      BB_G2_KS_AM19 : Bool;   // Belebung - SigmaControl Gebläse 2 - Alarme - Ansaugdruck p1 zu niedrig -> Verschmutzung des Ansaugfilters
      BB_G2_KS_AM20 : Bool;   // Belebung - SigmaControl Gebläse 2 - Alarme - Temperatur unter der Schalldämmhaube zu hoch
      BB_G2_KS_AM21 : Bool;   // Belebung - SigmaControl Gebläse 2 - Alarme - Reserve
      BB_G2_KS_AM22 : Bool;   // Belebung - SigmaControl Gebläse 2 - Alarme - Differenzdruck zu hoch
      BB_G2_KS_AM23 : Bool;   // Belebung - SigmaControl Gebläse 2 - Alarme - Ansaugtemperatur t1 zu hoch
      BB_G2_KS_AM24 : Bool;   // Belebung - SigmaControl Gebläse 2 - Alarme - Ansaugtemperatur t1 zu niedrig
      BB_G2_KS_AM41 : Bool;   // Belebung - SigmaControl Gebläse 2 - Alarme - Überspannung im Stromversorgungsnetz
      BB_G2_KS_AM42 : Bool;   // Belebung - SigmaControl Gebläse 2 - Alarme - Fehler am AFxM-Ventil-Aktor
      BB_G2_KS_AM43 : Bool;   // Belebung - SigmaControl Gebläse 2 - Alarme - Reserve
      BB_G2_KS_AM44 : Bool;   // Belebung - SigmaControl Gebläse 2 - Alarme - Blockdrehzahl liegt außerhalb des erlaubten Bereiches -> Fehler im Antriebsmotor oder Keilriemen
      BB_G2_KS_AM45 : Bool;   // Belebung - SigmaControl Gebläse 2 - Alarme - Vibration des Gebläses zu hoch
      BB_G2_KS_AM46 : Bool;   // Belebung - SigmaControl Gebläse 2 - Alarme - Interner Fehler Frequenzumrichter für Gebläsemotor
      BB_G2_KS_AM47 : Bool;   // Belebung - SigmaControl Gebläse 2 - Alarme - Kommunikationsfehler RS485-FC -> USS-Bus Kommunikationsfehler
      BB_G2_KS_AM48 : Bool;   // Belebung - SigmaControl Gebläse 2 - Alarme - Sammelmeldung des Leistungsteils FU
      BB_G2_KS_AM33 : Bool;   // Belebung - SigmaControl Gebläse 2 - Alarme - Reserve
      BB_G2_KS_AM34 : Bool;   // Belebung - SigmaControl Gebläse 2 - Alarme - Reserve
      BB_G2_KS_AM35 : Bool;   // Belebung - SigmaControl Gebläse 2 - Alarme - Druckdifferenz über den Block zu niedrig
      BB_G2_KS_AM36 : Bool;   // Belebung - SigmaControl Gebläse 2 - Alarme - Reserve
      BB_G2_KS_AM37 : Bool;   // Belebung - SigmaControl Gebläse 2 - Alarme - Reserve
      BB_G2_KS_AM38 : Bool;   // Belebung - SigmaControl Gebläse 2 - Alarme - Ansaugdruck p1 zu niedrig -> Verschmutzung des Ansaugfilters
      BB_G2_KS_AM39 : Bool;   // Belebung - SigmaControl Gebläse 2 - Alarme - Enddruck p2 zu hoch
      BB_G2_KS_AM40 : Bool;   // Belebung - SigmaControl Gebläse 2 - Alarme - Netzschütz schaltet nicht aus oder nicht ein
      BB_G2_KS_AM57 : Bool;   // Belebung - SigmaControl Gebläse 2 - Alarme - Schwerlastüberwachung ausgelöst FU -> Schwerlastüberwachung ausgelöst
      BB_G2_KS_AM58 : Bool;   // Belebung - SigmaControl Gebläse 2 - Alarme - p1-Sensor-Fehler Fehler Drucksensor Ansaugseite Gebläseblock
      BB_G2_KS_AM59 : Bool;   // Belebung - SigmaControl Gebläse 2 - Alarme - p2-Sensor-Fehler Fehler Drucksensor Auslassseite Gebläseblock
      BB_G2_KS_AM60 : Bool;   // Belebung - SigmaControl Gebläse 2 - Alarme - Fehler externer Analogeingang Fehler am externen Analogeingang
      BB_G2_KS_AM61 : Bool;   // Belebung - SigmaControl Gebläse 2 - Alarme - t2-Sensor-Fehler Fehler Sensor PT100 Auslasssseite Gebläseblock
      BB_G2_KS_AM62 : Bool;   // Belebung - SigmaControl Gebläse 2 - Alarme - t_S-Sensor-Fehler Fehler Sensor PT100 Schalldämmhaube
      BB_G2_KS_AM63 : Bool;   // Belebung - SigmaControl Gebläse 2 - Alarme - t1-Sensor-Fehler Fehler Sensor PT100 Ansaugseite Gebläseblock
      BB_G2_KS_AM64 : Bool;   // Belebung - SigmaControl Gebläse 2 - Alarme - t_M-Sensor-Fehler Fehler Sensor PT100 Antriebsmotor
      BB_G2_KS_AM49 : Bool;   // Belebung - SigmaControl Gebläse 2 - Alarme - Reserve
      BB_G2_KS_AM50 : Bool;   // Belebung - SigmaControl Gebläse 2 - Alarme - Nachschmiereinrichtung meldet seit längerer Zeit einen Fehler
      BB_G2_KS_AM51 : Bool;   // Belebung - SigmaControl Gebläse 2 - Alarme - Reserve
      BB_G2_KS_AM52 : Bool;   // Belebung - SigmaControl Gebläse 2 - Alarme - Reserve
      BB_G2_KS_AM53 : Bool;   // Belebung - SigmaControl Gebläse 2 - Alarme - Fehler USS Handler FU -> USS Busfehler
      BB_G2_KS_AM54 : Bool;   // Belebung - SigmaControl Gebläse 2 - Alarme - PKW-Anfragen erfolglos FU -> USS Kommunikation gestört
      BB_G2_KS_AM55 : Bool;   // Belebung - SigmaControl Gebläse 2 - Alarme - Fehler FU Einschaltung FU -> Fehler beim Einschalten des Frequenzumrichters
      BB_G2_KS_AM56 : Bool;   // Belebung - SigmaControl Gebläse 2 - Alarme - Motor -> n_min nicht erreicht FU -> Mindestdrehzahl nicht erreicht
      BB_G2_KS_AM73 : Bool;   // Belebung - SigmaControl Gebläse 2 - Alarme - Externe Meldung 1 Sammelmeldung externe Binärmeldung 1
      BB_G2_KS_AM74 : Bool;   // Belebung - SigmaControl Gebläse 2 - Alarme - Externe Meldung 2 Sammelmeldung externe Binärmeldung 2
      BB_G2_KS_AM75 : Bool;   // Belebung - SigmaControl Gebläse 2 - Alarme - Externe Meldung 3 Sammelmeldung externe Binärmeldung 3
      BB_G2_KS_AM76 : Bool;   // Belebung - SigmaControl Gebläse 2 - Alarme - Schalter p1 freier Schaltpunkt auf Druck p1
      BB_G2_KS_AM77 : Bool;   // Belebung - SigmaControl Gebläse 2 - Alarme - Schalter p2 freier Schaltpunkt auf Druck p2
      BB_G2_KS_AM78 : Bool;   // Belebung - SigmaControl Gebläse 2 - Alarme - Schalter T1 freier Schaltpunkt auf Temperatur T1
      BB_G2_KS_AM79 : Bool;   // Belebung - SigmaControl Gebläse 2 - Alarme - Schalter T2 freier Schaltpunkt auf Temperatur T2
      BB_G2_KS_AM80 : Bool;   // Belebung - SigmaControl Gebläse 2 - Alarme - Schalter Blockdrehzahl freier Schaltpunkt auf Blockdrehzahl
      BB_G2_KS_AM65 : Bool;   // Belebung - SigmaControl Gebläse 2 - Alarme - t3-Sensor-Fehler Fehler Sensor PT100 Öltemperatur
      BB_G2_KS_AM66 : Bool;   // Belebung - SigmaControl Gebläse 2 - Alarme - Reserve
      BB_G2_KS_AM67 : Bool;   // Belebung - SigmaControl Gebläse 2 - Alarme - Reserve
      BB_G2_KS_AM68 : Bool;   // Belebung - SigmaControl Gebläse 2 - Alarme - Reserve
      BB_G2_KS_AM69 : Bool;   // Belebung - SigmaControl Gebläse 2 - Alarme - Reserve
      BB_G2_KS_AM70 : Bool;   // Belebung - SigmaControl Gebläse 2 - Alarme - Schwingungsüberwachung VSE ? Schwingungen an Block oder Motor zu hoch
      BB_G2_KS_AM71 : Bool;   // Belebung - SigmaControl Gebläse 2 - Alarme - Schalter T3
      BB_G2_KS_AM72 : Bool;   // Belebung - SigmaControl Gebläse 2 - Alarme - Schalter T_S
      BB_G2_KS_WM9 : Bool;   // Belebung - SigmaControl Gebläse 2 - Warnungen - Temperatur unter der Schalldämmhaube zu hoch
      BB_G2_KS_WM10 : Bool;   // Belebung - SigmaControl Gebläse 2 - Warnungen - Umgebungstemperatur zu niedrig
      BB_G2_KS_WM11 : Bool;   // Belebung - SigmaControl Gebläse 2 - Warnungen - Differenzdruck zu hoch
      BB_G2_KS_WM12 : Bool;   // Belebung - SigmaControl Gebläse 2 - Warnungen - Differenzdruck zu niedrig
      BB_G2_KS_WM13 : Bool;   // Belebung - SigmaControl Gebläse 2 - Warnungen - Filter verstopft, Verschmutzung des Ansaugfilters
      BB_G2_KS_WM14 : Bool;   // Belebung - SigmaControl Gebläse 2 - Warnungen - Öltemperatur t3 zu hoch
      BB_G2_KS_WM15 : Bool;   // Belebung - SigmaControl Gebläse 2 - Warnungen - Com-Module Kommunikationsfehler Busankopplung über Com-Module ist unterbrochen
      BB_G2_KS_WM16 : Bool;   // Belebung - SigmaControl Gebläse 2 - Warnungen - SAM 4.0 Kommunikationsfehler Busankopplung über Com-Module ist unterbrochen
      BB_G2_KS_WM1 : Bool;   // Belebung - SigmaControl Gebläse 2 - Warnungen - Equipmentnummer unvollständig -> Equipmentnummer des Gebläses hat weniger als sieben Zeichen
      BB_G2_KS_WM2 : Bool;   // Belebung - SigmaControl Gebläse 2 - Warnungen - Sammelwarnung
      BB_G2_KS_WM3 : Bool;   // Belebung - SigmaControl Gebläse 2 - Warnungen - Reserve
      BB_G2_KS_WM4 : Bool;   // Belebung - SigmaControl Gebläse 2 - Warnungen - Schmierölstand Antriebsseite Gebläseblock zu niedrig
      BB_G2_KS_WM5 : Bool;   // Belebung - SigmaControl Gebläse 2 - Warnungen - Schmierölstand Steuerseite Gebläseblock zu niedrig
      BB_G2_KS_WM6 : Bool;   // Belebung - SigmaControl Gebläse 2 - Warnungen - Ansaugtemperatur t1 zu hoch
      BB_G2_KS_WM7 : Bool;   // Belebung - SigmaControl Gebläse 2 - Warnungen - Ansaugtemperatur t1 zu niedrig
      BB_G2_KS_WM8 : Bool;   // Belebung - SigmaControl Gebläse 2 - Warnungen - Verdichtungsendtemperatur t2 zu hoch
      BB_G2_KS_WM25 : Bool;   // Belebung - SigmaControl Gebläse 2 - Warnungen - Motorlager Schaltschrank-Lüfter -> Prüffrist abgelaufen
      BB_G2_KS_WM26 : Bool;   // Belebung - SigmaControl Gebläse 2 - Warnungen - Schmieröl -> Wartungsfrist abgelaufen
      BB_G2_KS_WM27 : Bool;   // Belebung - SigmaControl Gebläse 2 - Warnungen - Reserve
      BB_G2_KS_WM28 : Bool;   // Belebung - SigmaControl Gebläse 2 - Warnungen - Ansaugluftfilter -> Wartungsfrist abgelaufen
      BB_G2_KS_WM29 : Bool;   // Belebung - SigmaControl Gebläse 2 - Warnungen - Filtermatte -> Wartungsfrist abgelaufen
      BB_G2_KS_WM30 : Bool;   // Belebung - SigmaControl Gebläse 2 - Warnungen - Keilriemen -> Wartungsfrist abgelaufen
      BB_G2_KS_WM31 : Bool;   // Belebung - SigmaControl Gebläse 2 - Warnungen - Motorlager -> Wartungsfrist abgelaufen
      BB_G2_KS_WM32 : Bool;   // Belebung - SigmaControl Gebläse 2 - Warnungen - Motorlager Gebläsemotor -> Prüffrist abgelaufen
      BB_G2_KS_WM17 : Bool;   // Belebung - SigmaControl Gebläse 2 - Warnungen - Temperaturdifferenz t2 (VET) - t1 (Ansaugtemperatur) zu hoch
      BB_G2_KS_WM18 : Bool;   // Belebung - SigmaControl Gebläse 2 - Warnungen - Temperatur Gebläsemotor zu hoch
      BB_G2_KS_WM19 : Bool;   // Belebung - SigmaControl Gebläse 2 - Warnungen - Ansaugdruck p1 zu niedrig -> Verschmutzung des Ansaugfilters
      BB_G2_KS_WM20 : Bool;   // Belebung - SigmaControl Gebläse 2 - Warnungen - Enddruck p2 zu hoch
      BB_G2_KS_WM21 : Bool;   // Belebung - SigmaControl Gebläse 2 - Warnungen - Öltemperatur t3 zu niedrig
      BB_G2_KS_WM22 : Bool;   // Belebung - SigmaControl Gebläse 2 - Warnungen - Druckverhältnis über Block zu hoch
      BB_G2_KS_WM23 : Bool;   // Belebung - SigmaControl Gebläse 2 - Warnungen - Reserve
      BB_G2_KS_WM24 : Bool;   // Belebung - SigmaControl Gebläse 2 - Warnungen - maximale Schalthäufigkeit des Netzschützes ist erreicht -> austauschen
      BB_G2_KS_WM41 : Bool;   // Belebung - SigmaControl Gebläse 2 - Warnungen - Reserve
      BB_G2_KS_WM42 : Bool;   // Belebung - SigmaControl Gebläse 2 - Warnungen - Reserve
      BB_G2_KS_WM43 : Bool;   // Belebung - SigmaControl Gebläse 2 - Warnungen - Reserve
      BB_G2_KS_WM44 : Bool;   // Belebung - SigmaControl Gebläse 2 - Warnungen - Reserve
      BB_G2_KS_WM45 : Bool;   // Belebung - SigmaControl Gebläse 2 - Warnungen - Reserve
      BB_G2_KS_WM46 : Bool;   // Belebung - SigmaControl Gebläse 2 - Warnungen - Reserve
      BB_G2_KS_WM47 : Bool;   // Belebung - SigmaControl Gebläse 2 - Warnungen - Elektrobauteile und -installation -> Wartungsfrist abgelaufen
      BB_G2_KS_WM48 : Bool;   // Belebung - SigmaControl Gebläse 2 - Warnungen - Schmierung Motorlager Gebläsemotor -> Wartungsfrist abgelaufen
      BB_G2_KS_WM33 : Bool;   // Belebung - SigmaControl Gebläse 2 - Warnungen - Motorlager Schalldämmhauben-Lüfter -> Prüffrist abgelaufen
      BB_G2_KS_WM34 : Bool;   // Belebung - SigmaControl Gebläse 2 - Warnungen - FU-Lüfter -> Prüffrist abgelaufen
      BB_G2_KS_WM35 : Bool;   // Belebung - SigmaControl Gebläse 2 - Warnungen - Filter Getriebeentlüftung -> Wartungsfrist abgelaufen
      BB_G2_KS_WM36 : Bool;   // Belebung - SigmaControl Gebläse 2 - Warnungen - Maximal zulässige Schalthäufigkeit des Motors in den letzten 60 Minuten überschritten
      BB_G2_KS_WM37 : Bool;   // Belebung - SigmaControl Gebläse 2 - Warnungen - Reserve
      BB_G2_KS_WM38 : Bool;   // Belebung - SigmaControl Gebläse 2 - Warnungen - Ansaugdruck p1 zu niedrig -> Verschmutzung des Ansaugfilters
      BB_G2_KS_WM39 : Bool;   // Belebung - SigmaControl Gebläse 2 - Warnungen - Enddruck p2 zu hoch
      BB_G2_KS_WM40 : Bool;   // Belebung - SigmaControl Gebläse 2 - Warnungen - Überspannung im Stromversorgungsnetz
      BB_G2_KS_WM57 : Bool;   // Belebung - SigmaControl Gebläse 2 - Warnungen - Reserve
      BB_G2_KS_WM58 : Bool;   // Belebung - SigmaControl Gebläse 2 - Warnungen - SC2 zu SC2 Kommunikation unterbrochen
      BB_G2_KS_WM59 : Bool;   // Belebung - SigmaControl Gebläse 2 - Warnungen - Reserve
      BB_G2_KS_WM60 : Bool;   // Belebung - SigmaControl Gebläse 2 - Warnungen - Reserve
      BB_G2_KS_WM61 : Bool;   // Belebung - SigmaControl Gebläse 2 - Warnungen - Reserve
      BB_G2_KS_WM62 : Bool;   // Belebung - SigmaControl Gebläse 2 - Warnungen - FU im Servicebetrieb
      BB_G2_KS_WM63 : Bool;   // Belebung - SigmaControl Gebläse 2 - Warnungen - Test der "Safe Torque off" Abschaltpfade des Frequenzumrichters
      BB_G2_KS_WM64 : Bool;   // Belebung - SigmaControl Gebläse 2 - Warnungen - Reserve
      BB_G2_KS_WM49 : Bool;   // Belebung - SigmaControl Gebläse 2 - Warnungen - Jahreswartung fällig (erscheint 1 Jahr nach letzter Wartung)
      BB_G2_KS_WM50 : Bool;   // Belebung - SigmaControl Gebläse 2 - Warnungen - Fehler beim Schreiben der Daten auf SD-Karte
      BB_G2_KS_WM51 : Bool;   // Belebung - SigmaControl Gebläse 2 - Warnungen - Nachschmiereinrichtung meldet einen Fehler
      BB_G2_KS_WM52 : Bool;   // Belebung - SigmaControl Gebläse 2 - Warnungen - Reserve
      BB_G2_KS_WM53 : Bool;   // Belebung - SigmaControl Gebläse 2 - Warnungen - Reserve
      BB_G2_KS_WM54 : Bool;   // Belebung - SigmaControl Gebläse 2 - Warnungen - Reserve
      BB_G2_KS_WM55 : Bool;   // Belebung - SigmaControl Gebläse 2 - Warnungen - Reserve
      BB_G2_KS_WM56 : Bool;   // Belebung - SigmaControl Gebläse 2 - Warnungen - Reserve
      BB_G2_KS_WM73 : Bool;   // Belebung - SigmaControl Gebläse 2 - Warnungen - Sammelmeldung externe Binärmeldung 1
      BB_G2_KS_WM74 : Bool;   // Belebung - SigmaControl Gebläse 2 - Warnungen - Sammelmeldung externe Binärmeldung 2
      BB_G2_KS_WM75 : Bool;   // Belebung - SigmaControl Gebläse 2 - Warnungen - Sammelmeldung externe Binärmeldung 3
      BB_G2_KS_WM76 : Bool;   // Belebung - SigmaControl Gebläse 2 - Warnungen - Schalter p1 freier Schaltpunkt auf Druck p1
      BB_G2_KS_WM77 : Bool;   // Belebung - SigmaControl Gebläse 2 - Warnungen - Schalter p2 freier Schaltpunkt auf Druck p2
      BB_G2_KS_WM78 : Bool;   // Belebung - SigmaControl Gebläse 2 - Warnungen - Schalter T1 freier Schaltpunkt auf Temperatur T1
      BB_G2_KS_WM79 : Bool;   // Belebung - SigmaControl Gebläse 2 - Warnungen - Schalter T2 freier Schaltpunkt auf Temperatur T2
      BB_G2_KS_WM80 : Bool;   // Belebung - SigmaControl Gebläse 2 - Warnungen - Schalter Blockdrehzahl freier Schaltpunkt auf Blockdrehzahl
      BB_G2_KS_WM65 : Bool;   // Belebung - SigmaControl Gebläse 2 - Warnungen - Reserve
      BB_G2_KS_WM66 : Bool;   // Belebung - SigmaControl Gebläse 2 - Warnungen - Reserve
      BB_G2_KS_WM67 : Bool;   // Belebung - SigmaControl Gebläse 2 - Warnungen - Reserve
      BB_G2_KS_WM68 : Bool;   // Belebung - SigmaControl Gebläse 2 - Warnungen - Schalter T3
      BB_G2_KS_WM69 : Bool;   // Belebung - SigmaControl Gebläse 2 - Warnungen - Schalter T_S
      BB_G2_KS_WM70 : Bool;   // Belebung - SigmaControl Gebläse 2 - Warnungen - Schwingungsüberwachung VSE -> Schwingungen an Block oder Motor
      BB_G2_KS_WM71 : Bool;   // Belebung - SigmaControl Gebläse 2 - Warnungen - Schwingungsüberwachung VSE -> Schwingungen an Block oder Motor
      BB_G2_KS_WM72 : Bool;   // Belebung - SigmaControl Gebläse 2 - Warnungen - Schwingungsüberwachung Summensignal -> Schwingungen an Block oder Motor
      BB_G2_KS_OM9 : Bool;   // Belebung - SigmaControl Gebläse 2 - Betriebsmeldungen - Reserve
      BB_G2_KS_OM10 : Bool;   // Belebung - SigmaControl Gebläse 2 - Betriebsmeldungen - Reserve
      BB_G2_KS_OM11 : Bool;   // Belebung - SigmaControl Gebläse 2 - Betriebsmeldungen - Warten auf Kaltstart -> Temperaturen im Gebläse zu niedrig
      BB_G2_KS_OM12 : Bool;   // Belebung - SigmaControl Gebläse 2 - Betriebsmeldungen - Ölrücklauf vom Filter in die Ölräume gestartet
      BB_G2_KS_OM13 : Bool;   // Belebung - SigmaControl Gebläse 2 - Betriebsmeldungen - Ölmangel (Ölrücklauf abwarten, Ölstand zu niedrig)
      BB_G2_KS_OM14 : Bool;   // Belebung - SigmaControl Gebläse 2 - Betriebsmeldungen - Reserve
      BB_G2_KS_OM15 : Bool;   // Belebung - SigmaControl Gebläse 2 - Betriebsmeldungen - Reserve
      BB_G2_KS_OM16 : Bool;   // Belebung - SigmaControl Gebläse 2 - Betriebsmeldungen - Reserve
      BB_G2_KS_OM1 : Bool;   // Belebung - SigmaControl Gebläse 2 - Betriebsmeldungen - Reserve
      BB_G2_KS_OM2 : Bool;   // Belebung - SigmaControl Gebläse 2 - Betriebsmeldungen - Reserve
      BB_G2_KS_OM3 : Bool;   // Belebung - SigmaControl Gebläse 2 - Betriebsmeldungen - Reserve
      BB_G2_KS_OM4 : Bool;   // Belebung - SigmaControl Gebläse 2 - Betriebsmeldungen - Reserve
      BB_G2_KS_OM5 : Bool;   // Belebung - SigmaControl Gebläse 2 - Betriebsmeldungen - Reserve
      BB_G2_KS_OM6 : Bool;   // Belebung - SigmaControl Gebläse 2 - Betriebsmeldungen - Reserve
      BB_G2_KS_OM7 : Bool;   // Belebung - SigmaControl Gebläse 2 - Betriebsmeldungen - Reserve
      BB_G2_KS_OM8 : Bool;   // Belebung - SigmaControl Gebläse 2 - Betriebsmeldungen - Reserve
      BB_G2_KS_OM25 : Bool;   // Belebung - SigmaControl Gebläse 2 - Betriebsmeldungen - Reserve
      BB_G2_KS_OM26 : Bool;   // Belebung - SigmaControl Gebläse 2 - Betriebsmeldungen - Reserve
      BB_G2_KS_OM27 : Bool;   // Belebung - SigmaControl Gebläse 2 - Betriebsmeldungen - Power OFF -> ON Neustart der Steuerung erforderlich
      BB_G2_KS_OM28 : Bool;   // Belebung - SigmaControl Gebläse 2 - Betriebsmeldungen - Reserve
      BB_G2_KS_OM29 : Bool;   // Belebung - SigmaControl Gebläse 2 - Betriebsmeldungen - Reserve
      BB_G2_KS_OM30 : Bool;   // Belebung - SigmaControl Gebläse 2 - Betriebsmeldungen - Schalter p1 freier Schaltpunkt auf Druck p1
      BB_G2_KS_OM31 : Bool;   // Belebung - SigmaControl Gebläse 2 - Betriebsmeldungen - Schalter p2 freier Schaltpunkt auf Druck p2
      BB_G2_KS_OM32 : Bool;   // Belebung - SigmaControl Gebläse 2 - Betriebsmeldungen - Schalter T1 freier Schaltpunkt auf Temperatur T1
      BB_G2_KS_OM17 : Bool;   // Belebung - SigmaControl Gebläse 2 - Betriebsmeldungen - Externe Meldung 1 Sammelmeldung externe Binärmeldung 1
      BB_G2_KS_OM18 : Bool;   // Belebung - SigmaControl Gebläse 2 - Betriebsmeldungen - Externe Meldung 2 Sammelmeldung externe Binärmeldung 2
      BB_G2_KS_OM19 : Bool;   // Belebung - SigmaControl Gebläse 2 - Betriebsmeldungen - Externe Meldung 3 Sammelmeldung externe Binärmeldung 3
      BB_G2_KS_OM20 : Bool;   // Belebung - SigmaControl Gebläse 2 - Betriebsmeldungen - Schwingungsüberwachung VSE -> Schwingungen an Block oder Motor
      BB_G2_KS_OM21 : Bool;   // Belebung - SigmaControl Gebläse 2 - Betriebsmeldungen - Schwingungsüberwachung Summensignal -> Schwingungen an Block oder Motor
      BB_G2_KS_OM22 : Bool;   // Belebung - SigmaControl Gebläse 2 - Betriebsmeldungen - Reserve
      BB_G2_KS_OM23 : Bool;   // Belebung - SigmaControl Gebläse 2 - Betriebsmeldungen - Reserve
      BB_G2_KS_OM24 : Bool;   // Belebung - SigmaControl Gebläse 2 - Betriebsmeldungen - Reserve
      BB_G2_KS_OM41 : Bool;   // Belebung - SigmaControl Gebläse 2 - Betriebsmeldungen - Reserve
      BB_G2_KS_OM42 : Bool;   // Belebung - SigmaControl Gebläse 2 - Betriebsmeldungen - Reserve
      BB_G2_KS_OM43 : Bool;   // Belebung - SigmaControl Gebläse 2 - Betriebsmeldungen - Reserve
      BB_G2_KS_OM44 : Bool;   // Belebung - SigmaControl Gebläse 2 - Betriebsmeldungen - Reserve
      BB_G2_KS_OM45 : Bool;   // Belebung - SigmaControl Gebläse 2 - Betriebsmeldungen - Reserve
      BB_G2_KS_OM46 : Bool;   // Belebung - SigmaControl Gebläse 2 - Betriebsmeldungen - Reserve
      BB_G2_KS_OM47 : Bool;   // Belebung - SigmaControl Gebläse 2 - Betriebsmeldungen - Reserve
      BB_G2_KS_OM48 : Bool;   // Belebung - SigmaControl Gebläse 2 - Betriebsmeldungen - Reserve
      BB_G2_KS_OM33 : Bool;   // Belebung - SigmaControl Gebläse 2 - Betriebsmeldungen - Schalter T2 freier Schaltpunkt auf Temperatur T2
      BB_G2_KS_OM34 : Bool;   // Belebung - SigmaControl Gebläse 2 - Betriebsmeldungen - Schalter Blockdrehzahl freier Schaltpunkt auf Blockdrehzahl
      BB_G2_KS_OM35 : Bool;   // Belebung - SigmaControl Gebläse 2 - Betriebsmeldungen - Schalter T3
      BB_G2_KS_OM36 : Bool;   // Belebung - SigmaControl Gebläse 2 - Betriebsmeldungen - Schalter T_S
      BB_G2_KS_OM37 : Bool;   // Belebung - SigmaControl Gebläse 2 - Betriebsmeldungen - Reserve
      BB_G2_KS_OM38 : Bool;   // Belebung - SigmaControl Gebläse 2 - Betriebsmeldungen - Ansaugdruck p1 zu niedrig -> Verschmutzung des Ansaugfilters
      BB_G2_KS_OM39 : Bool;   // Belebung - SigmaControl Gebläse 2 - Betriebsmeldungen - Enddruck p2 zu hoch
      BB_G2_KS_OM40 : Bool;   // Belebung - SigmaControl Gebläse 2 - Betriebsmeldungen - Techniker vor Ort Ein Techniker arbeitet an der Maschine
      BB_G2_KS_BS8 : Bool;   // Belebung - SigmaControl Gebläse 2 - Status - Reserve
      BB_G2_KS_BS9 : Bool;   // Belebung - SigmaControl Gebläse 2 - Status - Gebläse Ein (Maschine eingeschaltet)
      BB_G2_KS_BS10 : Bool;   // Belebung - SigmaControl Gebläse 2 - Status - Lüfter Nachkühler Betrieb
      BB_G2_KS_BS11 : Bool;   // Belebung - SigmaControl Gebläse 2 - Status - Lüfter Schalldämmhaube Betrieb
      BB_G2_KS_BS12 : Bool;   // Belebung - SigmaControl Gebläse 2 - Status - Reserve
      BB_G2_KS_BS13 : Bool;   // Belebung - SigmaControl Gebläse 2 - Status - Reserve
      BB_G2_KS_BS14 : Bool;   // Belebung - SigmaControl Gebläse 2 - Status - Sammelwartung
      BB_G2_KS_BS15 : Bool;   // Belebung - SigmaControl Gebläse 2 - Status - Sammelwarnung
      BB_G2_KS_BS0 : Bool;   // Belebung - SigmaControl Gebläse 2 - Status - Anlage Ein + Fernbetrieb Ein + Bus (Receive)
      BB_G2_KS_BS1 : Bool;   // Belebung - SigmaControl Gebläse 2 - Status - Motor Betrieb
      BB_G2_KS_BS2 : Bool;   // Belebung - SigmaControl Gebläse 2 - Status - Lastlauf
      BB_G2_KS_BS3 : Bool;   // Belebung - SigmaControl Gebläse 2 - Status - Leerlauf
      BB_G2_KS_BS4 : Bool;   // Belebung - SigmaControl Gebläse 2 - Status - vor-Ort Betrieb
      BB_G2_KS_BS5 : Bool;   // Belebung - SigmaControl Gebläse 2 - Status - Anlage Ein
      BB_G2_KS_BS6 : Bool;   // Belebung - SigmaControl Gebläse 2 - Status - Sammelstörung
      BB_G2_KS_BS7 : Bool;   // Belebung - SigmaControl Gebläse 2 - Status - Sammelwarnung/-warnung
      BB_G2_KS_BS24 : Bool;   // Belebung - SigmaControl Gebläse 2 - Status - Betriebsart Volumenstromregelung
      BB_G2_KS_BS25 : Bool;   // Belebung - SigmaControl Gebläse 2 - Status - Reserve
      BB_G2_KS_BS26 : Bool;   // Belebung - SigmaControl Gebläse 2 - Status - Reserve
      BB_G2_KS_BS27 : Bool;   // Belebung - SigmaControl Gebläse 2 - Status - Reserve
      BB_G2_KS_BS28 : Bool;   // Belebung - SigmaControl Gebläse 2 - Status - Reserve
      BB_G2_KS_BS29 : Bool;   // Belebung - SigmaControl Gebläse 2 - Status - Reserve
      BB_G2_KS_BS30 : Bool;   // Belebung - SigmaControl Gebläse 2 - Status - Reserve
      BB_G2_KS_BS31 : Bool;   // Belebung - SigmaControl Gebläse 2 - Status - Reserve
      BB_G2_KS_BS16 : Bool;   // Belebung - SigmaControl Gebläse 2 - Status - Modus "Gebläse Ein" nur durch vor-Ort-Bedienung
      BB_G2_KS_BS17 : Bool;   // Belebung - SigmaControl Gebläse 2 - Status - Reserve
      BB_G2_KS_BS18 : Bool;   // Belebung - SigmaControl Gebläse 2 - Status - Reserve
      BB_G2_KS_BS19 : Bool;   // Belebung - SigmaControl Gebläse 2 - Status - Reserve
      BB_G2_KS_BS20 : Bool;   // Belebung - SigmaControl Gebläse 2 - Status - Betriebsart Festdrehzahl
      BB_G2_KS_BS21 : Bool;   // Belebung - SigmaControl Gebläse 2 - Status - Betriebsart externe Drehzahlvorgabe
      BB_G2_KS_BS22 : Bool;   // Belebung - SigmaControl Gebläse 2 - Status - Betriebsart Druckregelung
      BB_G2_KS_BS23 : Bool;   // Belebung - SigmaControl Gebläse 2 - Status - Betriebsart externe Größe
      BB_G2_KS_BS40 : Bool;   // Belebung - SigmaControl Gebläse 2 - Status - Reserve
      BB_G2_KS_BS41 : Bool;   // Belebung - SigmaControl Gebläse 2 - Status - Reserve
      BB_G2_KS_BS42 : Bool;   // Belebung - SigmaControl Gebläse 2 - Status - Reserve
      BB_G2_KS_BS43 : Bool;   // Belebung - SigmaControl Gebläse 2 - Status - Reserve
      BB_G2_KS_BS44 : Bool;   // Belebung - SigmaControl Gebläse 2 - Status - Reserve
      BB_G2_KS_BS45 : Bool;   // Belebung - SigmaControl Gebläse 2 - Status - Reserve
      BB_G2_KS_BS46 : Bool;   // Belebung - SigmaControl Gebläse 2 - Status - Reserve
      BB_G2_KS_BS47 : Bool;   // Belebung - SigmaControl Gebläse 2 - Status - Reserve
      BB_G2_KS_BS32 : Bool;   // Belebung - SigmaControl Gebläse 2 - Status - Reserve
      BB_G2_KS_BS33 : Bool;   // Belebung - SigmaControl Gebläse 2 - Status - Reserve
      BB_G2_KS_BS34 : Bool;   // Belebung - SigmaControl Gebläse 2 - Status - Reserve
      BB_G2_KS_BS35 : Bool;   // Belebung - SigmaControl Gebläse 2 - Status - Reserve
      BB_G2_KS_BS36 : Bool;   // Belebung - SigmaControl Gebläse 2 - Status - Modus Laststeuerung Lastsignal durch ext. Kontakt ist aktiv
      BB_G2_KS_BS37 : Bool;   // Belebung - SigmaControl Gebläse 2 - Status - Reserve
      BB_G2_KS_BS38 : Bool;   // Belebung - SigmaControl Gebläse 2 - Status - Modus Laststeuerung Lastsignal durch BusMaster ist aktiv
      BB_G2_KS_BS39 : Bool;   // Belebung - SigmaControl Gebläse 2 - Status - Reserve
      BB_G2_KS_BS56 : Bool;   // Belebung - SigmaControl Gebläse 2 - Status - Reserve
      BB_G2_KS_BS57 : Bool;   // Belebung - SigmaControl Gebläse 2 - Status - Reserve
      BB_G2_KS_BS58 : Bool;   // Belebung - SigmaControl Gebläse 2 - Status - Reserve
      BB_G2_KS_BS59 : Bool;   // Belebung - SigmaControl Gebläse 2 - Status - Reserve
      BB_G2_KS_BS60 : Bool;   // Belebung - SigmaControl Gebläse 2 - Status - Reserve
      BB_G2_KS_BS61 : Bool;   // Belebung - SigmaControl Gebläse 2 - Status - Reserve
      BB_G2_KS_BS62 : Bool;   // Belebung - SigmaControl Gebläse 2 - Status - Reserve
      BB_G2_KS_BS63 : Bool;   // Belebung - SigmaControl Gebläse 2 - Status - Reserve
      BB_G2_KS_BS48 : Bool;   // Belebung - SigmaControl Gebläse 2 - Status - Reserve
      BB_G2_KS_BS49 : Bool;   // Belebung - SigmaControl Gebläse 2 - Status - Reserve
      BB_G2_KS_BS50 : Bool;   // Belebung - SigmaControl Gebläse 2 - Status - Reserve
      BB_G2_KS_BS51 : Bool;   // Belebung - SigmaControl Gebläse 2 - Status - Automatischer Anlauf nach Netzspannung EIN
      BB_G2_KS_BS52 : Bool;   // Belebung - SigmaControl Gebläse 2 - Status - Reserve
      BB_G2_KS_BS53 : Bool;   // Belebung - SigmaControl Gebläse 2 - Status - Reserve
      BB_G2_KS_BS54 : Bool;   // Belebung - SigmaControl Gebläse 2 - Status - Reserve
      BB_G2_KS_BS55 : Bool;   // Belebung - SigmaControl Gebläse 2 - Status - Meldungs-Quittierung durch Master
      BB_G3_KS_AM9 : Bool;   // Belebung - SigmaControl Gebläse 3 - Alarme - Zulässige Innentemperatur von SIGMA CONTROL 2 MCS oder IOM überschritten
      BB_G3_KS_AM10 : Bool;   // Belebung - SigmaControl Gebläse 3 - Alarme - Enddruck p2 zu hoch
      BB_G3_KS_AM11 : Bool;   // Belebung - SigmaControl Gebläse 3 - Alarme - Reserve
      BB_G3_KS_AM12 : Bool;   // Belebung - SigmaControl Gebläse 3 - Alarme - Reserve
      BB_G3_KS_AM13 : Bool;   // Belebung - SigmaControl Gebläse 3 - Alarme - Überlast Gebläsemotor -> Abschaltung wegen Überlastung
      BB_G3_KS_AM14 : Bool;   // Belebung - SigmaControl Gebläse 3 - Alarme - Abschaltung des Nachkühler-Lüfters wegen Überlastung
      BB_G3_KS_AM15 : Bool;   // Belebung - SigmaControl Gebläse 3 - Alarme - Maximal zulässige Verdichtungs-Endtemperatur (VET) überschritten
      BB_G3_KS_AM16 : Bool;   // Belebung - SigmaControl Gebläse 3 - Alarme - Reserve
      BB_G3_KS_AM1 : Bool;   // Belebung - SigmaControl Gebläse 3 - Alarme - Reserve
      BB_G3_KS_AM2 : Bool;   // Belebung - SigmaControl Gebläse 3 - Alarme - Temperatur Gebläsemotor zu hoch
      BB_G3_KS_AM3 : Bool;   // Belebung - SigmaControl Gebläse 3 - Alarme - Reserve
      BB_G3_KS_AM4 : Bool;   // Belebung - SigmaControl Gebläse 3 - Alarme - NOT-HALT-Befehlsgerät betätigt
      BB_G3_KS_AM5 : Bool;   // Belebung - SigmaControl Gebläse 3 - Alarme - Schmierölstand Antriebsseite Gebläseblock zu niedrig
      BB_G3_KS_AM6 : Bool;   // Belebung - SigmaControl Gebläse 3 - Alarme - Schmierölstand Steuerseite Gebläseblock zu niedrig
      BB_G3_KS_AM7 : Bool;   // Belebung - SigmaControl Gebläse 3 - Alarme - Phasenfehler oder Unter-/Überspannung Gebläsemotor
      BB_G3_KS_AM8 : Bool;   // Belebung - SigmaControl Gebläse 3 - Alarme - Diagnose-Sammelmeldung
      BB_G3_KS_AM25 : Bool;   // Belebung - SigmaControl Gebläse 3 - Alarme - Sammelfehler IOM
      BB_G3_KS_AM26 : Bool;   // Belebung - SigmaControl Gebläse 3 - Alarme - Reserve
      BB_G3_KS_AM27 : Bool;   // Belebung - SigmaControl Gebläse 3 - Alarme - Filter verstopft -> Verschmutzung des Ansaugfilters
      BB_G3_KS_AM28 : Bool;   // Belebung - SigmaControl Gebläse 3 - Alarme - Öltemperatur t3 sehr hoch
      BB_G3_KS_AM29 : Bool;   // Belebung - SigmaControl Gebläse 3 - Alarme - Reserve
      BB_G3_KS_AM30 : Bool;   // Belebung - SigmaControl Gebläse 3 - Alarme - Reserve
      BB_G3_KS_AM31 : Bool;   // Belebung - SigmaControl Gebläse 3 - Alarme - Temperaturdifferenz t2 (VET) - t1 (Ansaugtemperatur) zu hoch
      BB_G3_KS_AM32 : Bool;   // Belebung - SigmaControl Gebläse 3 - Alarme - Druckverhältnis über Block zu hoch
      BB_G3_KS_AM17 : Bool;   // Belebung - SigmaControl Gebläse 3 - Alarme - Reserve
      BB_G3_KS_AM18 : Bool;   // Belebung - SigmaControl Gebläse 3 - Alarme - Abschaltung des Schalldämmhauben-Lüfters wegen Überlastung
      BB_G3_KS_AM19 : Bool;   // Belebung - SigmaControl Gebläse 3 - Alarme - Ansaugdruck p1 zu niedrig -> Verschmutzung des Ansaugfilters
      BB_G3_KS_AM20 : Bool;   // Belebung - SigmaControl Gebläse 3 - Alarme - Temperatur unter der Schalldämmhaube zu hoch
      BB_G3_KS_AM21 : Bool;   // Belebung - SigmaControl Gebläse 3 - Alarme - Reserve
      BB_G3_KS_AM22 : Bool;   // Belebung - SigmaControl Gebläse 3 - Alarme - Differenzdruck zu hoch
      BB_G3_KS_AM23 : Bool;   // Belebung - SigmaControl Gebläse 3 - Alarme - Ansaugtemperatur t1 zu hoch
      BB_G3_KS_AM24 : Bool;   // Belebung - SigmaControl Gebläse 3 - Alarme - Ansaugtemperatur t1 zu niedrig
      BB_G3_KS_AM41 : Bool;   // Belebung - SigmaControl Gebläse 3 - Alarme - Überspannung im Stromversorgungsnetz
      BB_G3_KS_AM42 : Bool;   // Belebung - SigmaControl Gebläse 3 - Alarme - Fehler am AFxM-Ventil-Aktor
      BB_G3_KS_AM43 : Bool;   // Belebung - SigmaControl Gebläse 3 - Alarme - Reserve
      BB_G3_KS_AM44 : Bool;   // Belebung - SigmaControl Gebläse 3 - Alarme - Blockdrehzahl liegt außerhalb des erlaubten Bereiches -> Fehler im Antriebsmotor oder Keilriemen
      BB_G3_KS_AM45 : Bool;   // Belebung - SigmaControl Gebläse 3 - Alarme - Vibration des Gebläses zu hoch
      BB_G3_KS_AM46 : Bool;   // Belebung - SigmaControl Gebläse 3 - Alarme - Interner Fehler Frequenzumrichter für Gebläsemotor
      BB_G3_KS_AM47 : Bool;   // Belebung - SigmaControl Gebläse 3 - Alarme - Kommunikationsfehler RS485-FC -> USS-Bus Kommunikationsfehler
      BB_G3_KS_AM48 : Bool;   // Belebung - SigmaControl Gebläse 3 - Alarme - Sammelmeldung des Leistungsteils FU
      BB_G3_KS_AM33 : Bool;   // Belebung - SigmaControl Gebläse 3 - Alarme - Reserve
      BB_G3_KS_AM34 : Bool;   // Belebung - SigmaControl Gebläse 3 - Alarme - Reserve
      BB_G3_KS_AM35 : Bool;   // Belebung - SigmaControl Gebläse 3 - Alarme - Druckdifferenz über den Block zu niedrig
      BB_G3_KS_AM36 : Bool;   // Belebung - SigmaControl Gebläse 3 - Alarme - Reserve
      BB_G3_KS_AM37 : Bool;   // Belebung - SigmaControl Gebläse 3 - Alarme - Reserve
      BB_G3_KS_AM38 : Bool;   // Belebung - SigmaControl Gebläse 3 - Alarme - Ansaugdruck p1 zu niedrig -> Verschmutzung des Ansaugfilters
      BB_G3_KS_AM39 : Bool;   // Belebung - SigmaControl Gebläse 3 - Alarme - Enddruck p2 zu hoch
      BB_G3_KS_AM40 : Bool;   // Belebung - SigmaControl Gebläse 3 - Alarme - Netzschütz schaltet nicht aus oder nicht ein
      BB_G3_KS_AM57 : Bool;   // Belebung - SigmaControl Gebläse 3 - Alarme - Schwerlastüberwachung ausgelöst FU -> Schwerlastüberwachung ausgelöst
      BB_G3_KS_AM58 : Bool;   // Belebung - SigmaControl Gebläse 3 - Alarme - p1-Sensor-Fehler Fehler Drucksensor Ansaugseite Gebläseblock
      BB_G3_KS_AM59 : Bool;   // Belebung - SigmaControl Gebläse 3 - Alarme - p2-Sensor-Fehler Fehler Drucksensor Auslassseite Gebläseblock
      BB_G3_KS_AM60 : Bool;   // Belebung - SigmaControl Gebläse 3 - Alarme - Fehler externer Analogeingang Fehler am externen Analogeingang
      BB_G3_KS_AM61 : Bool;   // Belebung - SigmaControl Gebläse 3 - Alarme - t2-Sensor-Fehler Fehler Sensor PT100 Auslasssseite Gebläseblock
      BB_G3_KS_AM62 : Bool;   // Belebung - SigmaControl Gebläse 3 - Alarme - t_S-Sensor-Fehler Fehler Sensor PT100 Schalldämmhaube
      BB_G3_KS_AM63 : Bool;   // Belebung - SigmaControl Gebläse 3 - Alarme - t1-Sensor-Fehler Fehler Sensor PT100 Ansaugseite Gebläseblock
      BB_G3_KS_AM64 : Bool;   // Belebung - SigmaControl Gebläse 3 - Alarme - t_M-Sensor-Fehler Fehler Sensor PT100 Antriebsmotor
      BB_G3_KS_AM49 : Bool;   // Belebung - SigmaControl Gebläse 3 - Alarme - Reserve
      BB_G3_KS_AM50 : Bool;   // Belebung - SigmaControl Gebläse 3 - Alarme - Nachschmiereinrichtung meldet seit längerer Zeit einen Fehler
      BB_G3_KS_AM51 : Bool;   // Belebung - SigmaControl Gebläse 3 - Alarme - Reserve
      BB_G3_KS_AM52 : Bool;   // Belebung - SigmaControl Gebläse 3 - Alarme - Reserve
      BB_G3_KS_AM53 : Bool;   // Belebung - SigmaControl Gebläse 3 - Alarme - Fehler USS Handler FU -> USS Busfehler
      BB_G3_KS_AM54 : Bool;   // Belebung - SigmaControl Gebläse 3 - Alarme - PKW-Anfragen erfolglos FU -> USS Kommunikation gestört
      BB_G3_KS_AM55 : Bool;   // Belebung - SigmaControl Gebläse 3 - Alarme - Fehler FU Einschaltung FU -> Fehler beim Einschalten des Frequenzumrichters
      BB_G3_KS_AM56 : Bool;   // Belebung - SigmaControl Gebläse 3 - Alarme - Motor -> n_min nicht erreicht FU -> Mindestdrehzahl nicht erreicht
      BB_G3_KS_AM73 : Bool;   // Belebung - SigmaControl Gebläse 3 - Alarme - Externe Meldung 1 Sammelmeldung externe Binärmeldung 1
      BB_G3_KS_AM74 : Bool;   // Belebung - SigmaControl Gebläse 3 - Alarme - Externe Meldung 2 Sammelmeldung externe Binärmeldung 2
      BB_G3_KS_AM75 : Bool;   // Belebung - SigmaControl Gebläse 3 - Alarme - Externe Meldung 3 Sammelmeldung externe Binärmeldung 3
      BB_G3_KS_AM76 : Bool;   // Belebung - SigmaControl Gebläse 3 - Alarme - Schalter p1 freier Schaltpunkt auf Druck p1
      BB_G3_KS_AM77 : Bool;   // Belebung - SigmaControl Gebläse 3 - Alarme - Schalter p2 freier Schaltpunkt auf Druck p2
      BB_G3_KS_AM78 : Bool;   // Belebung - SigmaControl Gebläse 3 - Alarme - Schalter T1 freier Schaltpunkt auf Temperatur T1
      BB_G3_KS_AM79 : Bool;   // Belebung - SigmaControl Gebläse 3 - Alarme - Schalter T2 freier Schaltpunkt auf Temperatur T2
      BB_G3_KS_AM80 : Bool;   // Belebung - SigmaControl Gebläse 3 - Alarme - Schalter Blockdrehzahl freier Schaltpunkt auf Blockdrehzahl
      BB_G3_KS_AM65 : Bool;   // Belebung - SigmaControl Gebläse 3 - Alarme - t3-Sensor-Fehler Fehler Sensor PT100 Öltemperatur
      BB_G3_KS_AM66 : Bool;   // Belebung - SigmaControl Gebläse 3 - Alarme - Reserve
      BB_G3_KS_AM67 : Bool;   // Belebung - SigmaControl Gebläse 3 - Alarme - Reserve
      BB_G3_KS_AM68 : Bool;   // Belebung - SigmaControl Gebläse 3 - Alarme - Reserve
      BB_G3_KS_AM69 : Bool;   // Belebung - SigmaControl Gebläse 3 - Alarme - Reserve
      BB_G3_KS_AM70 : Bool;   // Belebung - SigmaControl Gebläse 3 - Alarme - Schwingungsüberwachung VSE ? Schwingungen an Block oder Motor zu hoch
      BB_G3_KS_AM71 : Bool;   // Belebung - SigmaControl Gebläse 3 - Alarme - Schalter T3
      BB_G3_KS_AM72 : Bool;   // Belebung - SigmaControl Gebläse 3 - Alarme - Schalter T_S
      BB_G3_KS_WM9 : Bool;   // Belebung - SigmaControl Gebläse 3 - Warnungen - Temperatur unter der Schalldämmhaube zu hoch
      BB_G3_KS_WM10 : Bool;   // Belebung - SigmaControl Gebläse 3 - Warnungen - Umgebungstemperatur zu niedrig
      BB_G3_KS_WM11 : Bool;   // Belebung - SigmaControl Gebläse 3 - Warnungen - Differenzdruck zu hoch
      BB_G3_KS_WM12 : Bool;   // Belebung - SigmaControl Gebläse 3 - Warnungen - Differenzdruck zu niedrig
      BB_G3_KS_WM13 : Bool;   // Belebung - SigmaControl Gebläse 3 - Warnungen - Filter verstopft, Verschmutzung des Ansaugfilters
      BB_G3_KS_WM14 : Bool;   // Belebung - SigmaControl Gebläse 3 - Warnungen - Öltemperatur t3 zu hoch
      BB_G3_KS_WM15 : Bool;   // Belebung - SigmaControl Gebläse 3 - Warnungen - Com-Module Kommunikationsfehler Busankopplung über Com-Module ist unterbrochen
      BB_G3_KS_WM16 : Bool;   // Belebung - SigmaControl Gebläse 3 - Warnungen - SAM 4.0 Kommunikationsfehler Busankopplung über Com-Module ist unterbrochen
      BB_G3_KS_WM1 : Bool;   // Belebung - SigmaControl Gebläse 3 - Warnungen - Equipmentnummer unvollständig -> Equipmentnummer des Gebläses hat weniger als sieben Zeichen
      BB_G3_KS_WM2 : Bool;   // Belebung - SigmaControl Gebläse 3 - Warnungen - Sammelwarnung
      BB_G3_KS_WM3 : Bool;   // Belebung - SigmaControl Gebläse 3 - Warnungen - Reserve
      BB_G3_KS_WM4 : Bool;   // Belebung - SigmaControl Gebläse 3 - Warnungen - Schmierölstand Antriebsseite Gebläseblock zu niedrig
      BB_G3_KS_WM5 : Bool;   // Belebung - SigmaControl Gebläse 3 - Warnungen - Schmierölstand Steuerseite Gebläseblock zu niedrig
      BB_G3_KS_WM6 : Bool;   // Belebung - SigmaControl Gebläse 3 - Warnungen - Ansaugtemperatur t1 zu hoch
      BB_G3_KS_WM7 : Bool;   // Belebung - SigmaControl Gebläse 3 - Warnungen - Ansaugtemperatur t1 zu niedrig
      BB_G3_KS_WM8 : Bool;   // Belebung - SigmaControl Gebläse 3 - Warnungen - Verdichtungsendtemperatur t2 zu hoch
      BB_G3_KS_WM25 : Bool;   // Belebung - SigmaControl Gebläse 3 - Warnungen - Motorlager Schaltschrank-Lüfter -> Prüffrist abgelaufen
      BB_G3_KS_WM26 : Bool;   // Belebung - SigmaControl Gebläse 3 - Warnungen - Schmieröl -> Wartungsfrist abgelaufen
      BB_G3_KS_WM27 : Bool;   // Belebung - SigmaControl Gebläse 3 - Warnungen - Reserve
      BB_G3_KS_WM28 : Bool;   // Belebung - SigmaControl Gebläse 3 - Warnungen - Ansaugluftfilter -> Wartungsfrist abgelaufen
      BB_G3_KS_WM29 : Bool;   // Belebung - SigmaControl Gebläse 3 - Warnungen - Filtermatte -> Wartungsfrist abgelaufen
      BB_G3_KS_WM30 : Bool;   // Belebung - SigmaControl Gebläse 3 - Warnungen - Keilriemen -> Wartungsfrist abgelaufen
      BB_G3_KS_WM31 : Bool;   // Belebung - SigmaControl Gebläse 3 - Warnungen - Motorlager -> Wartungsfrist abgelaufen
      BB_G3_KS_WM32 : Bool;   // Belebung - SigmaControl Gebläse 3 - Warnungen - Motorlager Gebläsemotor -> Prüffrist abgelaufen
      BB_G3_KS_WM17 : Bool;   // Belebung - SigmaControl Gebläse 3 - Warnungen - Temperaturdifferenz t2 (VET) - t1 (Ansaugtemperatur) zu hoch
      BB_G3_KS_WM18 : Bool;   // Belebung - SigmaControl Gebläse 3 - Warnungen - Temperatur Gebläsemotor zu hoch
      BB_G3_KS_WM19 : Bool;   // Belebung - SigmaControl Gebläse 3 - Warnungen - Ansaugdruck p1 zu niedrig -> Verschmutzung des Ansaugfilters
      BB_G3_KS_WM20 : Bool;   // Belebung - SigmaControl Gebläse 3 - Warnungen - Enddruck p2 zu hoch
      BB_G3_KS_WM21 : Bool;   // Belebung - SigmaControl Gebläse 3 - Warnungen - Öltemperatur t3 zu niedrig
      BB_G3_KS_WM22 : Bool;   // Belebung - SigmaControl Gebläse 3 - Warnungen - Druckverhältnis über Block zu hoch
      BB_G3_KS_WM23 : Bool;   // Belebung - SigmaControl Gebläse 3 - Warnungen - Reserve
      BB_G3_KS_WM24 : Bool;   // Belebung - SigmaControl Gebläse 3 - Warnungen - maximale Schalthäufigkeit des Netzschützes ist erreicht -> austauschen
      BB_G3_KS_WM41 : Bool;   // Belebung - SigmaControl Gebläse 3 - Warnungen - Reserve
      BB_G3_KS_WM42 : Bool;   // Belebung - SigmaControl Gebläse 3 - Warnungen - Reserve
      BB_G3_KS_WM43 : Bool;   // Belebung - SigmaControl Gebläse 3 - Warnungen - Reserve
      BB_G3_KS_WM44 : Bool;   // Belebung - SigmaControl Gebläse 3 - Warnungen - Reserve
      BB_G3_KS_WM45 : Bool;   // Belebung - SigmaControl Gebläse 3 - Warnungen - Reserve
      BB_G3_KS_WM46 : Bool;   // Belebung - SigmaControl Gebläse 3 - Warnungen - Reserve
      BB_G3_KS_WM47 : Bool;   // Belebung - SigmaControl Gebläse 3 - Warnungen - Elektrobauteile und -installation -> Wartungsfrist abgelaufen
      BB_G3_KS_WM48 : Bool;   // Belebung - SigmaControl Gebläse 3 - Warnungen - Schmierung Motorlager Gebläsemotor -> Wartungsfrist abgelaufen
      BB_G3_KS_WM33 : Bool;   // Belebung - SigmaControl Gebläse 3 - Warnungen - Motorlager Schalldämmhauben-Lüfter -> Prüffrist abgelaufen
      BB_G3_KS_WM34 : Bool;   // Belebung - SigmaControl Gebläse 3 - Warnungen - FU-Lüfter -> Prüffrist abgelaufen
      BB_G3_KS_WM35 : Bool;   // Belebung - SigmaControl Gebläse 3 - Warnungen - Filter Getriebeentlüftung -> Wartungsfrist abgelaufen
      BB_G3_KS_WM36 : Bool;   // Belebung - SigmaControl Gebläse 3 - Warnungen - Maximal zulässige Schalthäufigkeit des Motors in den letzten 60 Minuten überschritten
      BB_G3_KS_WM37 : Bool;   // Belebung - SigmaControl Gebläse 3 - Warnungen - Reserve
      BB_G3_KS_WM38 : Bool;   // Belebung - SigmaControl Gebläse 3 - Warnungen - Ansaugdruck p1 zu niedrig -> Verschmutzung des Ansaugfilters
      BB_G3_KS_WM39 : Bool;   // Belebung - SigmaControl Gebläse 3 - Warnungen - Enddruck p2 zu hoch
      BB_G3_KS_WM40 : Bool;   // Belebung - SigmaControl Gebläse 3 - Warnungen - Überspannung im Stromversorgungsnetz
      BB_G3_KS_WM57 : Bool;   // Belebung - SigmaControl Gebläse 3 - Warnungen - Reserve
      BB_G3_KS_WM58 : Bool;   // Belebung - SigmaControl Gebläse 3 - Warnungen - SC2 zu SC2 Kommunikation unterbrochen
      BB_G3_KS_WM59 : Bool;   // Belebung - SigmaControl Gebläse 3 - Warnungen - Reserve
      BB_G3_KS_WM60 : Bool;   // Belebung - SigmaControl Gebläse 3 - Warnungen - Reserve
      BB_G3_KS_WM61 : Bool;   // Belebung - SigmaControl Gebläse 3 - Warnungen - Reserve
      BB_G3_KS_WM62 : Bool;   // Belebung - SigmaControl Gebläse 3 - Warnungen - FU im Servicebetrieb
      BB_G3_KS_WM63 : Bool;   // Belebung - SigmaControl Gebläse 3 - Warnungen - Test der "Safe Torque off" Abschaltpfade des Frequenzumrichters
      BB_G3_KS_WM64 : Bool;   // Belebung - SigmaControl Gebläse 3 - Warnungen - Reserve
      BB_G3_KS_WM49 : Bool;   // Belebung - SigmaControl Gebläse 3 - Warnungen - Jahreswartung fällig (erscheint 1 Jahr nach letzter Wartung)
      BB_G3_KS_WM50 : Bool;   // Belebung - SigmaControl Gebläse 3 - Warnungen - Fehler beim Schreiben der Daten auf SD-Karte
      BB_G3_KS_WM51 : Bool;   // Belebung - SigmaControl Gebläse 3 - Warnungen - Nachschmiereinrichtung meldet einen Fehler
      BB_G3_KS_WM52 : Bool;   // Belebung - SigmaControl Gebläse 3 - Warnungen - Reserve
      BB_G3_KS_WM53 : Bool;   // Belebung - SigmaControl Gebläse 3 - Warnungen - Reserve
      BB_G3_KS_WM54 : Bool;   // Belebung - SigmaControl Gebläse 3 - Warnungen - Reserve
      BB_G3_KS_WM55 : Bool;   // Belebung - SigmaControl Gebläse 3 - Warnungen - Reserve
      BB_G3_KS_WM56 : Bool;   // Belebung - SigmaControl Gebläse 3 - Warnungen - Reserve
      BB_G3_KS_WM73 : Bool;   // Belebung - SigmaControl Gebläse 3 - Warnungen - Sammelmeldung externe Binärmeldung 1
      BB_G3_KS_WM74 : Bool;   // Belebung - SigmaControl Gebläse 3 - Warnungen - Sammelmeldung externe Binärmeldung 2
      BB_G3_KS_WM75 : Bool;   // Belebung - SigmaControl Gebläse 3 - Warnungen - Sammelmeldung externe Binärmeldung 3
      BB_G3_KS_WM76 : Bool;   // Belebung - SigmaControl Gebläse 3 - Warnungen - Schalter p1 freier Schaltpunkt auf Druck p1
      BB_G3_KS_WM77 : Bool;   // Belebung - SigmaControl Gebläse 3 - Warnungen - Schalter p2 freier Schaltpunkt auf Druck p2
      BB_G3_KS_WM78 : Bool;   // Belebung - SigmaControl Gebläse 3 - Warnungen - Schalter T1 freier Schaltpunkt auf Temperatur T1
      BB_G3_KS_WM79 : Bool;   // Belebung - SigmaControl Gebläse 3 - Warnungen - Schalter T2 freier Schaltpunkt auf Temperatur T2
      BB_G3_KS_WM80 : Bool;   // Belebung - SigmaControl Gebläse 3 - Warnungen - Schalter Blockdrehzahl freier Schaltpunkt auf Blockdrehzahl
      BB_G3_KS_WM65 : Bool;   // Belebung - SigmaControl Gebläse 3 - Warnungen - Reserve
      BB_G3_KS_WM66 : Bool;   // Belebung - SigmaControl Gebläse 3 - Warnungen - Reserve
      BB_G3_KS_WM67 : Bool;   // Belebung - SigmaControl Gebläse 3 - Warnungen - Reserve
      BB_G3_KS_WM68 : Bool;   // Belebung - SigmaControl Gebläse 3 - Warnungen - Schalter T3
      BB_G3_KS_WM69 : Bool;   // Belebung - SigmaControl Gebläse 3 - Warnungen - Schalter T_S
      BB_G3_KS_WM70 : Bool;   // Belebung - SigmaControl Gebläse 3 - Warnungen - Schwingungsüberwachung VSE -> Schwingungen an Block oder Motor
      BB_G3_KS_WM71 : Bool;   // Belebung - SigmaControl Gebläse 3 - Warnungen - Schwingungsüberwachung VSE -> Schwingungen an Block oder Motor
      BB_G3_KS_WM72 : Bool;   // Belebung - SigmaControl Gebläse 3 - Warnungen - Schwingungsüberwachung Summensignal -> Schwingungen an Block oder Motor
      BB_G3_KS_OM9 : Bool;   // Belebung - SigmaControl Gebläse 3 - Betriebsmeldungen - Reserve
      BB_G3_KS_OM10 : Bool;   // Belebung - SigmaControl Gebläse 3 - Betriebsmeldungen - Reserve
      BB_G3_KS_OM11 : Bool;   // Belebung - SigmaControl Gebläse 3 - Betriebsmeldungen - Warten auf Kaltstart -> Temperaturen im Gebläse zu niedrig
      BB_G3_KS_OM12 : Bool;   // Belebung - SigmaControl Gebläse 3 - Betriebsmeldungen - Ölrücklauf vom Filter in die Ölräume gestartet
      BB_G3_KS_OM13 : Bool;   // Belebung - SigmaControl Gebläse 3 - Betriebsmeldungen - Ölmangel (Ölrücklauf abwarten, Ölstand zu niedrig)
      BB_G3_KS_OM14 : Bool;   // Belebung - SigmaControl Gebläse 3 - Betriebsmeldungen - Reserve
      BB_G3_KS_OM15 : Bool;   // Belebung - SigmaControl Gebläse 3 - Betriebsmeldungen - Reserve
      BB_G3_KS_OM16 : Bool;   // Belebung - SigmaControl Gebläse 3 - Betriebsmeldungen - Reserve
      BB_G3_KS_OM1 : Bool;   // Belebung - SigmaControl Gebläse 3 - Betriebsmeldungen - Reserve
      BB_G3_KS_OM2 : Bool;   // Belebung - SigmaControl Gebläse 3 - Betriebsmeldungen - Reserve
      BB_G3_KS_OM3 : Bool;   // Belebung - SigmaControl Gebläse 3 - Betriebsmeldungen - Reserve
      BB_G3_KS_OM4 : Bool;   // Belebung - SigmaControl Gebläse 3 - Betriebsmeldungen - Reserve
      BB_G3_KS_OM5 : Bool;   // Belebung - SigmaControl Gebläse 3 - Betriebsmeldungen - Reserve
      BB_G3_KS_OM6 : Bool;   // Belebung - SigmaControl Gebläse 3 - Betriebsmeldungen - Reserve
      BB_G3_KS_OM7 : Bool;   // Belebung - SigmaControl Gebläse 3 - Betriebsmeldungen - Reserve
      BB_G3_KS_OM8 : Bool;   // Belebung - SigmaControl Gebläse 3 - Betriebsmeldungen - Reserve
      BB_G3_KS_OM25 : Bool;   // Belebung - SigmaControl Gebläse 3 - Betriebsmeldungen - Reserve
      BB_G3_KS_OM26 : Bool;   // Belebung - SigmaControl Gebläse 3 - Betriebsmeldungen - Reserve
      BB_G3_KS_OM27 : Bool;   // Belebung - SigmaControl Gebläse 3 - Betriebsmeldungen - Power OFF -> ON Neustart der Steuerung erforderlich
      BB_G3_KS_OM28 : Bool;   // Belebung - SigmaControl Gebläse 3 - Betriebsmeldungen - Reserve
      BB_G3_KS_OM29 : Bool;   // Belebung - SigmaControl Gebläse 3 - Betriebsmeldungen - Reserve
      BB_G3_KS_OM30 : Bool;   // Belebung - SigmaControl Gebläse 3 - Betriebsmeldungen - Schalter p1 freier Schaltpunkt auf Druck p1
      BB_G3_KS_OM31 : Bool;   // Belebung - SigmaControl Gebläse 3 - Betriebsmeldungen - Schalter p2 freier Schaltpunkt auf Druck p2
      BB_G3_KS_OM32 : Bool;   // Belebung - SigmaControl Gebläse 3 - Betriebsmeldungen - Schalter T1 freier Schaltpunkt auf Temperatur T1
      BB_G3_KS_OM17 : Bool;   // Belebung - SigmaControl Gebläse 3 - Betriebsmeldungen - Externe Meldung 1 Sammelmeldung externe Binärmeldung 1
      BB_G3_KS_OM18 : Bool;   // Belebung - SigmaControl Gebläse 3 - Betriebsmeldungen - Externe Meldung 2 Sammelmeldung externe Binärmeldung 2
      BB_G3_KS_OM19 : Bool;   // Belebung - SigmaControl Gebläse 3 - Betriebsmeldungen - Externe Meldung 3 Sammelmeldung externe Binärmeldung 3
      BB_G3_KS_OM20 : Bool;   // Belebung - SigmaControl Gebläse 3 - Betriebsmeldungen - Schwingungsüberwachung VSE -> Schwingungen an Block oder Motor
      BB_G3_KS_OM21 : Bool;   // Belebung - SigmaControl Gebläse 3 - Betriebsmeldungen - Schwingungsüberwachung Summensignal -> Schwingungen an Block oder Motor
      BB_G3_KS_OM22 : Bool;   // Belebung - SigmaControl Gebläse 3 - Betriebsmeldungen - Reserve
      BB_G3_KS_OM23 : Bool;   // Belebung - SigmaControl Gebläse 3 - Betriebsmeldungen - Reserve
      BB_G3_KS_OM24 : Bool;   // Belebung - SigmaControl Gebläse 3 - Betriebsmeldungen - Reserve
      BB_G3_KS_OM41 : Bool;   // Belebung - SigmaControl Gebläse 3 - Betriebsmeldungen - Reserve
      BB_G3_KS_OM42 : Bool;   // Belebung - SigmaControl Gebläse 3 - Betriebsmeldungen - Reserve
      BB_G3_KS_OM43 : Bool;   // Belebung - SigmaControl Gebläse 3 - Betriebsmeldungen - Reserve
      BB_G3_KS_OM44 : Bool;   // Belebung - SigmaControl Gebläse 3 - Betriebsmeldungen - Reserve
      BB_G3_KS_OM45 : Bool;   // Belebung - SigmaControl Gebläse 3 - Betriebsmeldungen - Reserve
      BB_G3_KS_OM46 : Bool;   // Belebung - SigmaControl Gebläse 3 - Betriebsmeldungen - Reserve
      BB_G3_KS_OM47 : Bool;   // Belebung - SigmaControl Gebläse 3 - Betriebsmeldungen - Reserve
      BB_G3_KS_OM48 : Bool;   // Belebung - SigmaControl Gebläse 3 - Betriebsmeldungen - Reserve
      BB_G3_KS_OM33 : Bool;   // Belebung - SigmaControl Gebläse 3 - Betriebsmeldungen - Schalter T2 freier Schaltpunkt auf Temperatur T2
      BB_G3_KS_OM34 : Bool;   // Belebung - SigmaControl Gebläse 3 - Betriebsmeldungen - Schalter Blockdrehzahl freier Schaltpunkt auf Blockdrehzahl
      BB_G3_KS_OM35 : Bool;   // Belebung - SigmaControl Gebläse 3 - Betriebsmeldungen - Schalter T3
      BB_G3_KS_OM36 : Bool;   // Belebung - SigmaControl Gebläse 3 - Betriebsmeldungen - Schalter T_S
      BB_G3_KS_OM37 : Bool;   // Belebung - SigmaControl Gebläse 3 - Betriebsmeldungen - Reserve
      BB_G3_KS_OM38 : Bool;   // Belebung - SigmaControl Gebläse 3 - Betriebsmeldungen - Ansaugdruck p1 zu niedrig -> Verschmutzung des Ansaugfilters
      BB_G3_KS_OM39 : Bool;   // Belebung - SigmaControl Gebläse 3 - Betriebsmeldungen - Enddruck p2 zu hoch
      BB_G3_KS_OM40 : Bool;   // Belebung - SigmaControl Gebläse 3 - Betriebsmeldungen - Techniker vor Ort Ein Techniker arbeitet an der Maschine
      BB_G3_KS_BS8 : Bool;   // Belebung - SigmaControl Gebläse 3 - Status - Reserve
      BB_G3_KS_BS9 : Bool;   // Belebung - SigmaControl Gebläse 3 - Status - Gebläse Ein (Maschine eingeschaltet)
      BB_G3_KS_BS10 : Bool;   // Belebung - SigmaControl Gebläse 3 - Status - Lüfter Nachkühler Betrieb
      BB_G3_KS_BS11 : Bool;   // Belebung - SigmaControl Gebläse 3 - Status - Lüfter Schalldämmhaube Betrieb
      BB_G3_KS_BS12 : Bool;   // Belebung - SigmaControl Gebläse 3 - Status - Reserve
      BB_G3_KS_BS13 : Bool;   // Belebung - SigmaControl Gebläse 3 - Status - Reserve
      BB_G3_KS_BS14 : Bool;   // Belebung - SigmaControl Gebläse 3 - Status - Sammelwartung
      BB_G3_KS_BS15 : Bool;   // Belebung - SigmaControl Gebläse 3 - Status - Sammelwarnung
      BB_G3_KS_BS0 : Bool;   // Belebung - SigmaControl Gebläse 3 - Status - Anlage Ein + Fernbetrieb Ein + Bus (Receive)
      BB_G3_KS_BS1 : Bool;   // Belebung - SigmaControl Gebläse 3 - Status - Motor Betrieb
      BB_G3_KS_BS2 : Bool;   // Belebung - SigmaControl Gebläse 3 - Status - Lastlauf
      BB_G3_KS_BS3 : Bool;   // Belebung - SigmaControl Gebläse 3 - Status - Leerlauf
      BB_G3_KS_BS4 : Bool;   // Belebung - SigmaControl Gebläse 3 - Status - vor-Ort Betrieb
      BB_G3_KS_BS5 : Bool;   // Belebung - SigmaControl Gebläse 3 - Status - Anlage Ein
      BB_G3_KS_BS6 : Bool;   // Belebung - SigmaControl Gebläse 3 - Status - Sammelstörung
      BB_G3_KS_BS7 : Bool;   // Belebung - SigmaControl Gebläse 3 - Status - Sammelwarnung/-warnung
      BB_G3_KS_BS24 : Bool;   // Belebung - SigmaControl Gebläse 3 - Status - Betriebsart Volumenstromregelung
      BB_G3_KS_BS25 : Bool;   // Belebung - SigmaControl Gebläse 3 - Status - Reserve
      BB_G3_KS_BS26 : Bool;   // Belebung - SigmaControl Gebläse 3 - Status - Reserve
      BB_G3_KS_BS27 : Bool;   // Belebung - SigmaControl Gebläse 3 - Status - Reserve
      BB_G3_KS_BS28 : Bool;   // Belebung - SigmaControl Gebläse 3 - Status - Reserve
      BB_G3_KS_BS29 : Bool;   // Belebung - SigmaControl Gebläse 3 - Status - Reserve
      BB_G3_KS_BS30 : Bool;   // Belebung - SigmaControl Gebläse 3 - Status - Reserve
      BB_G3_KS_BS31 : Bool;   // Belebung - SigmaControl Gebläse 3 - Status - Reserve
      BB_G3_KS_BS16 : Bool;   // Belebung - SigmaControl Gebläse 3 - Status - Modus "Gebläse Ein" nur durch vor-Ort-Bedienung
      BB_G3_KS_BS17 : Bool;   // Belebung - SigmaControl Gebläse 3 - Status - Reserve
      BB_G3_KS_BS18 : Bool;   // Belebung - SigmaControl Gebläse 3 - Status - Reserve
      BB_G3_KS_BS19 : Bool;   // Belebung - SigmaControl Gebläse 3 - Status - Reserve
      BB_G3_KS_BS20 : Bool;   // Belebung - SigmaControl Gebläse 3 - Status - Betriebsart Festdrehzahl
      BB_G3_KS_BS21 : Bool;   // Belebung - SigmaControl Gebläse 3 - Status - Betriebsart externe Drehzahlvorgabe
      BB_G3_KS_BS22 : Bool;   // Belebung - SigmaControl Gebläse 3 - Status - Betriebsart Druckregelung
      BB_G3_KS_BS23 : Bool;   // Belebung - SigmaControl Gebläse 3 - Status - Betriebsart externe Größe
      BB_G3_KS_BS40 : Bool;   // Belebung - SigmaControl Gebläse 3 - Status - Reserve
      BB_G3_KS_BS41 : Bool;   // Belebung - SigmaControl Gebläse 3 - Status - Reserve
      BB_G3_KS_BS42 : Bool;   // Belebung - SigmaControl Gebläse 3 - Status - Reserve
      BB_G3_KS_BS43 : Bool;   // Belebung - SigmaControl Gebläse 3 - Status - Reserve
      BB_G3_KS_BS44 : Bool;   // Belebung - SigmaControl Gebläse 3 - Status - Reserve
      BB_G3_KS_BS45 : Bool;   // Belebung - SigmaControl Gebläse 3 - Status - Reserve
      BB_G3_KS_BS46 : Bool;   // Belebung - SigmaControl Gebläse 3 - Status - Reserve
      BB_G3_KS_BS47 : Bool;   // Belebung - SigmaControl Gebläse 3 - Status - Reserve
      BB_G3_KS_BS32 : Bool;   // Belebung - SigmaControl Gebläse 3 - Status - Reserve
      BB_G3_KS_BS33 : Bool;   // Belebung - SigmaControl Gebläse 3 - Status - Reserve
      BB_G3_KS_BS34 : Bool;   // Belebung - SigmaControl Gebläse 3 - Status - Reserve
      BB_G3_KS_BS35 : Bool;   // Belebung - SigmaControl Gebläse 3 - Status - Reserve
      BB_G3_KS_BS36 : Bool;   // Belebung - SigmaControl Gebläse 3 - Status - Modus Laststeuerung Lastsignal durch ext. Kontakt ist aktiv
      BB_G3_KS_BS37 : Bool;   // Belebung - SigmaControl Gebläse 3 - Status - Reserve
      BB_G3_KS_BS38 : Bool;   // Belebung - SigmaControl Gebläse 3 - Status - Modus Laststeuerung Lastsignal durch BusMaster ist aktiv
      BB_G3_KS_BS39 : Bool;   // Belebung - SigmaControl Gebläse 3 - Status - Reserve
      BB_G3_KS_BS56 : Bool;   // Belebung - SigmaControl Gebläse 3 - Status - Reserve
      BB_G3_KS_BS57 : Bool;   // Belebung - SigmaControl Gebläse 3 - Status - Reserve
      BB_G3_KS_BS58 : Bool;   // Belebung - SigmaControl Gebläse 3 - Status - Reserve
      BB_G3_KS_BS59 : Bool;   // Belebung - SigmaControl Gebläse 3 - Status - Reserve
      BB_G3_KS_BS60 : Bool;   // Belebung - SigmaControl Gebläse 3 - Status - Reserve
      BB_G3_KS_BS61 : Bool;   // Belebung - SigmaControl Gebläse 3 - Status - Reserve
      BB_G3_KS_BS62 : Bool;   // Belebung - SigmaControl Gebläse 3 - Status - Reserve
      BB_G3_KS_BS63 : Bool;   // Belebung - SigmaControl Gebläse 3 - Status - Reserve
      BB_G3_KS_BS48 : Bool;   // Belebung - SigmaControl Gebläse 3 - Status - Reserve
      BB_G3_KS_BS49 : Bool;   // Belebung - SigmaControl Gebläse 3 - Status - Reserve
      BB_G3_KS_BS50 : Bool;   // Belebung - SigmaControl Gebläse 3 - Status - Reserve
      BB_G3_KS_BS51 : Bool;   // Belebung - SigmaControl Gebläse 3 - Status - Automatischer Anlauf nach Netzspannung EIN
      BB_G3_KS_BS52 : Bool;   // Belebung - SigmaControl Gebläse 3 - Status - Reserve
      BB_G3_KS_BS53 : Bool;   // Belebung - SigmaControl Gebläse 3 - Status - Reserve
      BB_G3_KS_BS54 : Bool;   // Belebung - SigmaControl Gebläse 3 - Status - Reserve
      BB_G3_KS_BS55 : Bool;   // Belebung - SigmaControl Gebläse 3 - Status - Meldungs-Quittierung durch Master
      UPSStatus_BF_Bit00 : Bool;   // USV-Anlage - Status - Reserve
      UPSStatus_BF_Bit01 : Bool;   // USV-Anlage - Status - Netzbetrieb
      UPSStatus_BF_Bit02 : Bool;   // USV-Anlage - Status - Batteriebetrieb
      UPSStatus_BF_Bit03 : Bool;   // USV-Anlage - Status - Bypassbetrieb
      UPSStatus_BF_Bit04 : Bool;   // USV-Anlage - Status - Ausgang abgeschaltet
      UPSStatus_BF_Bit05 : Bool;   // USV-Anlage - Status - Sammelmeldung anstehend
      UPSStatus_BF_Bit06 : Bool;   // USV-Anlage - Status - Störung Eingang/Netzspannung
      UPSStatus_BF_Bit07 : Bool;   // USV-Anlage - Status - Test aktiv
      UPSStatus_BF_Bit08 : Bool;   // USV-Anlage - Status - Anforderung Zuschaltung
      UPSStatus_BF_Bit09 : Bool;   // USV-Anlage - Status - Abschaltung möglich, Restzeit prüfen!
      UPSStatus_BF_Bit10 : Bool;   // USV-Anlage - Status - Bypassbetrieb nach Befehl
      UPSStatus_BF_Bit11 : Bool;   // USV-Anlage - Status - Reserve
      UPSStatus_BF_Bit12 : Bool;   // USV-Anlage - Status - Reserve
      UPSStatus_BF_Bit13 : Bool;   // USV-Anlage - Status - ECO-Mode aktiv
      UPSStatus_BF_Bit14 : Bool;   // USV-Anlage - Status - Alarm/Information anstehend
      UPSStatus_BF_Bit15 : Bool;   // USV-Anlage - Status - Anlage in Störung
      UPSStatus_BF_Bit16 : Bool;   // USV-Anlage - Status - Reserve
      UPSStatus_BF_Bit17 : Bool;   // USV-Anlage - Status - Reserve
      UPSStatus_BF_Bit18 : Bool;   // USV-Anlage - Status - Reserve
      UPSStatus_BF_Bit19 : Bool;   // USV-Anlage - Status - Einspeisung gestört
      UPSStatus_BF_Bit20 : Bool;   // USV-Anlage - Status - Recovery-Mode nach Fehler
      UPSStatus_BF_Bit21 : Bool;   // USV-Anlage - Status - Überlast
      UPSStatus_BF_Bit22 : Bool;   // USV-Anlage - Status - Wartung aktiv
      UPSStatus_BF_Bit23 : Bool;   // USV-Anlage - Status - Effizienztest aktiv
      UPSStatus_BF_Bit24 : Bool;   // USV-Anlage - Status - Reserve
      UPSStatus_BF_Bit25 : Bool;   // USV-Anlage - Status - Reserve
      UPSStatus_BF_Bit26 : Bool;   // USV-Anlage - Status - Reserve
      UPSStatus_BF_Bit27 : Bool;   // USV-Anlage - Status - Reserve
      UPSStatus_BF_Bit28 : Bool;   // USV-Anlage - Status - Reserve
      UPSStatus_BF_Bit29 : Bool;   // USV-Anlage - Status - Reserve
      UPSStatus_BF_Bit30 : Bool;   // USV-Anlage - Status - Reserve
      UPSStatus_BF_Bit31 : Bool;   // USV-Anlage - Status - Reserve
      SimpleSignalingStatus_BF_Bit00 : Bool;   // USV-Anlage - Status - Störung Netzspannung
      SimpleSignalingStatus_BF_Bit01 : Bool;   // USV-Anlage - Status - Abschaltung steht unmittelbar bevor!
      SimpleSignalingStatus_BF_Bit02 : Bool;   // USV-Anlage - Status - Reserve
      SimpleSignalingStatus_BF_Bit03 : Bool;   // USV-Anlage - Status - Reserve
      SimpleSignalingStatus_BF_Bit04 : Bool;   // USV-Anlage - Status - Reserve
      SimpleSignalingStatus_BF_Bit05 : Bool;   // USV-Anlage - Status - Reserve
      SimpleSignalingStatus_BF_Bit06 : Bool;   // USV-Anlage - Status - Reserve
      SimpleSignalingStatus_BF_Bit07 : Bool;   // USV-Anlage - Status - Reserve
      SimpleSignalingStatus_BF_Bit08 : Bool;   // USV-Anlage - Status - Reserve
      SimpleSignalingStatus_BF_Bit09 : Bool;   // USV-Anlage - Status - Reserve
      SimpleSignalingStatus_BF_Bit10 : Bool;   // USV-Anlage - Status - Reserve
      SimpleSignalingStatus_BF_Bit11 : Bool;   // USV-Anlage - Status - Reserve
      SimpleSignalingStatus_BF_Bit12 : Bool;   // USV-Anlage - Status - Reserve
      SimpleSignalingStatus_BF_Bit13 : Bool;   // USV-Anlage - Status - Reserve
      SimpleSignalingStatus_BF_Bit14 : Bool;   // USV-Anlage - Status - Reserve
      SimpleSignalingStatus_BF_Bit15 : Bool;   // USV-Anlage - Status - Reserve
      UPSStatus_SF_Msg01 : Bool;   // USV-Anlage - Status - Sammelmeldung Fehler Hardware/intern
      UPSStatus_SF_Msg02 : Bool;   // USV-Anlage - Status - Sammelmeldung Fehler Powersystem
      UPSStatus_SF_Msg03 : Bool;   // USV-Anlage - Status - Sammelmeldung Fehler Batterie
      UPSStatus_SF_Msg04 : Bool;   // USV-Anlage - Status - Reserve
      UPSStatus_SF_Msg05 : Bool;   // USV-Anlage - Status - Reserve
      UPSStatus_SF_Msg06 : Bool;   // USV-Anlage - Status - Reserve
      UPSStatus_SF_Msg07 : Bool;   // USV-Anlage - Status - Reserve
      UPSStatus_SF_Msg08 : Bool;   // USV-Anlage - Status - Störung Kommunikation Modbus/TCP
      RES : Array[0..9] of Byte;
   END_STRUCT;


BEGIN
   E_Zulauf_AR_P1_Ein := FALSE;
   E_Zulauf_AR_P1_St := FALSE;
   E_Zulauf_AR_SS := FALSE;
   E_Zulauf_AR_P2_Ein := FALSE;
   E_Zulauf_AR_P2_St := FALSE;
   E_Zulauf_AR_HW := FALSE;
   E_Zulauf_AR_Niv_St := FALSE;
   E_Zulauf_AR_DF_ZI := FALSE;
   E_Zulauf_AR_DF_St := FALSE;
   E_Ablauf_pH_St := FALSE;
   E_Ablauf_O2_St := FALSE;
   E_Ablauf_DF_ZI := FALSE;
   E_Ablauf_DF_St := FALSE;
   E_BB_UeSS_DF_ZI := FALSE;
   E_ZEN_Res_1_6 := FALSE;
   E_ZEN_Res_1_7 := FALSE;
   E_NSHV_SS1_St := FALSE;
   E_NSHV_SS2_St := FALSE;
   E_NSHV_N02_AF_St := FALSE;
   E_NSHV_N03_AF_St := FALSE;
   E_NSHV_N04_AF_St := FALSE;
   E_NSHV_LS_Aus := FALSE;
   E_NSHV_LS_St := FALSE;
   E_NSHV_NA := FALSE;
   E_ZEN_Res_3_0 := FALSE;
   E_ZEN_Res_3_1 := FALSE;
   E_ZEN_Res_3_2 := FALSE;
   E_ZEN_Res_3_3 := FALSE;
   E_ZEN_Res_3_4 := FALSE;
   E_ZEN_Res_3_5 := FALSE;
   E_ZEN_Res_3_6 := FALSE;
   E_ZEN_Res_3_7 := FALSE;
   E_BB_G1_Ein := TRUE;
   E_BB_G1_St := FALSE;
   E_BB_G1_Bed_vOrt := FALSE;
   E_BB_G1_Bed_Fern := TRUE;
   E_BB_G1_AF_St := FALSE;
   E_BB_SHL_G1_Ein := TRUE;
   E_BB_SHL_G1_St := FALSE;
   E_BB_G2_Ein := TRUE;
   E_BB_G2_St := FALSE;
   E_BB_G2_Bed_vOrt := FALSE;
   E_BB_G2_Bed_Fern := TRUE;
   E_BB_G2_AF_St := FALSE;
   E_BB_SHL_G2_Ein := TRUE;
   E_BB_SHL_G2_St := FALSE;
   E_BB_G3_Ein := FALSE;
   E_BB_G3_St := FALSE;
   E_BB_G3_Bed_vOrt := FALSE;
   E_BB_G3_Bed_Fern := TRUE;
   E_BB_G3_AF_St := FALSE;
   E_BB_SHL_G3_Ein := FALSE;
   E_BB_SHL_G3_St := FALSE;
   E_BB_AV_Ein := FALSE;
   E_BB_AV_St := FALSE;
   E_BB_AV_AF_St := FALSE;
   E_BB_RT := FALSE;
   E_BB1_SR_K_Ein := FALSE;
   E_BB1_SR_K_St := FALSE;
   E_BB1_SR_K_AF_St := FALSE;
   E_BB_LS1_EA := FALSE;
   E_BB_LS1_EZ := TRUE;
   E_BB_LS1_St := FALSE;
   E_BB_LS1_Bed_vOrt := FALSE;
   E_BB_LS1_Bed_Fern := TRUE;
   E_BB_LS1_AF_St := FALSE;
   E_BB_LS2_EA := FALSE;
   E_BB_LS2_EZ := TRUE;
   E_BB_LS2_St := FALSE;
   E_BB_LS2_Bed_vOrt := FALSE;
   E_BB_LS2_Bed_Fern := TRUE;
   E_BB_LS2_AF_St := FALSE;
   E_BB1_RZP1_Ein := FALSE;
   E_BB1_RZP1_St := FALSE;
   E_BB1_RZP1_Bed_vOrt := FALSE;
   E_BB1_RZP1_Bed_Fern := TRUE;
   E_BB1_RZP1_AF_St := FALSE;
   E_BB1_RZP2_Ein := FALSE;
   E_BB1_RZP2_St := FALSE;
   E_BB1_RZP2_Bed_vOrt := FALSE;
   E_BB1_RZP2_Bed_Fern := TRUE;
   E_BB1_RZP2_AF_St := FALSE;
   E_BB1_UeSP_Ein := TRUE;
   E_BB1_UeSP_St := FALSE;
   E_BB1_UeSP_Bed_vOrt := FALSE;
   E_BB1_UeSP_Bed_Fern := TRUE;
   E_BB1_UeSP_AF_St := FALSE;
   E_BB1_AS1_EA := TRUE;
   E_BB1_AS1_EZ := FALSE;
   E_BB1_AS1_St := FALSE;
   E_BB1_AS1_Bed_vOrt := FALSE;
   E_BB1_AS1_Bed_Fern := TRUE;
   E_BB1_AS1_AF_St := FALSE;
   E_BB1_AS2_EA := FALSE;
   E_BB1_AS2_EZ := TRUE;
   E_BB1_AS2_St := FALSE;
   E_BB1_AS2_Bed_vOrt := FALSE;
   E_BB1_AS2_Bed_Fern := TRUE;
   E_BB1_AS2_AF_St := FALSE;
   E_BB1_SR1_Anst := FALSE;
   E_BB1_SR1_Bed_vOrt := FALSE;
   E_BB1_SR1_Bed_Fern := TRUE;
   E_BB1_SR1_AF_St := FALSE;
   E_BB1_SR2_Anst := FALSE;
   E_BB1_SR2_Bed_vOrt := FALSE;
   E_BB1_SR2_Bed_Fern := TRUE;
   E_BB1_SR2_AF_St := FALSE;
   E_BB1_O2_St := FALSE;
   E_BB1_DF_ZI := FALSE;
   E_BB1_DF_St := FALSE;
   E_BB2_RZP1_Ein := FALSE;
   E_BB2_RZP1_St := FALSE;
   E_BB2_RZP1_Bed_vOrt := FALSE;
   E_BB2_RZP1_Bed_Fern := TRUE;
   E_BB2_RZP1_AF_St := FALSE;
   E_BB2_RZP2_Ein := FALSE;
   E_BB2_RZP2_St := FALSE;
   E_BB2_RZP2_Bed_vOrt := FALSE;
   E_BB2_RZP2_Bed_Fern := TRUE;
   E_BB2_RZP2_AF_St := FALSE;
   E_BB2_UeSP_Ein := FALSE;
   E_BB2_UeSP_St := FALSE;
   E_BB2_UeSP_Bed_vOrt := FALSE;
   E_BB2_UeSP_Bed_Fern := TRUE;
   E_BB2_UeSP_AF_St := FALSE;
   E_BB2_AS1_EA := FALSE;
   E_BB2_AS1_EZ := TRUE;
   E_BB2_AS1_St := FALSE;
   E_BB2_AS1_Bed_vOrt := FALSE;
   E_BB2_AS1_Bed_Fern := TRUE;
   E_BB2_AS1_AF_St := FALSE;
   E_BB2_AS2_EA := TRUE;
   E_BB2_AS2_EZ := FALSE;
   E_BB2_AS2_St := FALSE;
   E_BB2_AS2_Bed_vOrt := FALSE;
   E_BB2_AS2_Bed_Fern := TRUE;
   E_BB2_AS2_AF_St := FALSE;
   E_BB2_SR1_Anst := FALSE;
   E_BB2_SR1_Bed_vOrt := FALSE;
   E_BB2_SR1_Bed_Fern := TRUE;
   E_BB2_SR1_AF_St := FALSE;
   E_BB2_SR2_Anst := FALSE;
   E_BB2_SR2_Bed_vOrt := FALSE;
   E_BB2_SR2_Bed_Fern := TRUE;
   E_BB2_SR2_AF_St := FALSE;
   E_BB2_O2_St := FALSE;
   E_BB2_DF_ZI := FALSE;
   E_BB2_DF_St := FALSE;
   E_BB2_SR_K_Ein := FALSE;
   E_BB2_SR_K_St := FALSE;
   E_BB2_SR_K_AF_St := FALSE;
   E_ZEN_Res_26_7 := FALSE;
   E_ZEN_Res_27_0 := FALSE;
   E_ZEN_Res_27_1 := FALSE;
   E_ZEN_Res_27_2 := FALSE;
   E_ZEN_Res_27_3 := FALSE;
   E_ZEN_Res_27_4 := FALSE;
   E_ZEN_Res_27_5 := FALSE;
   E_ZEN_Res_27_6 := FALSE;
   E_ZEN_Res_27_7 := FALSE;
   A_BB_G1_Ein := TRUE;
   A_BB_G2_Ein := TRUE;
   A_BB_G3_Ein := FALSE;
   A_BB_LS1_Auf := FALSE;
   A_BB_LS1_Zu := FALSE;
   A_BB_LS2_Auf := FALSE;
   A_BB_LS2_Zu := FALSE;
   A_ZEN_Res_12_7 := FALSE;
   A_BB1_RZP1_Ein := FALSE;
   A_BB1_RZP2_Ein := FALSE;
   A_BB1_UeSP_Ein := TRUE;
   A_BB1_AS1_Auf := FALSE;
   A_BB1_AS1_Zu := FALSE;
   A_BB1_AS2_Auf := FALSE;
   A_BB1_AS2_Zu := FALSE;
   A_BB1_SR1_Auf := FALSE;
   A_BB1_SR2_Auf := FALSE;
   A_ZEN_Res_14_1 := FALSE;
   A_ZEN_Res_14_2 := FALSE;
   A_ZEN_Res_14_3 := FALSE;
   A_ZEN_Res_14_4 := FALSE;
   A_ZEN_Res_14_5 := FALSE;
   A_ZEN_Res_14_6 := FALSE;
   A_ZEN_Res_14_7 := FALSE;
   A_BB2_RZP1_Ein := FALSE;
   A_BB2_RZP2_Ein := FALSE;
   A_BB2_UeSP_Ein := FALSE;
   A_BB2_AS1_Auf := FALSE;
   A_BB2_AS1_Zu := FALSE;
   A_BB2_AS2_Auf := FALSE;
   A_BB2_AS2_Zu := FALSE;
   A_BB2_SR1_Auf := FALSE;
   A_BB2_SR2_Auf := FALSE;
   A_ZEN_Res_16_1 := FALSE;
   A_ZEN_Res_16_2 := FALSE;
   A_ZEN_Res_16_3 := FALSE;
   A_ZEN_Res_16_4 := FALSE;
   A_ZEN_Res_16_5 := FALSE;
   A_ZEN_Res_16_6 := FALSE;
   A_ZEN_Res_16_7 := FALSE;
   A_Zulauf_AS_Auf := FALSE;
   A_Zulauf_AS_Zu := FALSE;
   A_ZEN_Res_17_2 := FALSE;
   A_ZEN_Res_17_3 := FALSE;
   A_ZEN_Res_17_4 := FALSE;
   A_ZEN_Res_17_5 := FALSE;
   A_ZEN_Res_17_6 := FALSE;
   A_ZEN_Res_17_7 := FALSE;
   E_Zulauf_RA_SA_Ein := TRUE;
   E_Zulauf_RA_HZS_Ein := FALSE;
   E_Zulauf_RA_VKS_Ein := FALSE;
   E_Zulauf_RA_V_Ein := TRUE;
   E_Zulauf_RA_RP_Ein := FALSE;
   E_Zulauf_RA_FP_Ein := FALSE;
   E_Zulauf_RA_SA_St := FALSE;
   E_Zulauf_RA_HZS_St := FALSE;
   E_Zulauf_RA_VKS_St := FALSE;
   E_Zulauf_RA_V_St := FALSE;
   E_Zulauf_RA_RP_St := FALSE;
   E_Zulauf_RA_FP_St := FALSE;
   E_Zulauf_RA_24V_St := FALSE;
   E_Zulauf_RA_US_St := FALSE;
   E_Zulauf_RA_230V_St := FALSE;
   E_Zulauf_DF_ZI := FALSE;
   E_Zulauf_DF_St := FALSE;
   E_Zulauf_Niv_St := FALSE;
   E_Verteiler_pH_St := FALSE;
   E_Zulauf_AS_EA := FALSE;
   E_Zulauf_AS_EZ := FALSE;
   E_Zulauf_AS_St := FALSE;
   E_Zulauf_AS_Bed_vOrt := FALSE;
   E_Zulauf_AS_Bed_Fern := TRUE;
   E_Zulauf_AS_AF_St := TRUE;
   E_ZEN_Res_31_1 := FALSE;
   E_ZEN_Res_31_2 := FALSE;
   E_ZEN_Res_31_3 := FALSE;
   E_ZEN_Res_31_4 := FALSE;
   E_ZEN_Res_31_5 := FALSE;
   E_ZEN_Res_31_6 := FALSE;
   E_ZEN_Res_31_7 := FALSE;
   E_ZEN_Res_40_0 := TRUE;
   E_Schlamm_BP_Ein := FALSE;
   E_Schlamm_BP_St := FALSE;
   E_Schlamm_BP_Bed_vOrt := FALSE;
   E_Schlamm_BP_Bed_Fern := TRUE;
   E_Schlamm_BP_AF_St := FALSE;
   E_Truebwasser_P1_Ein := FALSE;
   E_Truebwasser_P1_St := FALSE;
   E_Truebwasser_P1_Bed_vOrt := FALSE;
   E_Truebwasser_P1_Bed_Fern := TRUE;
   E_Truebwasser_P1_AF_St := FALSE;
   E_Truebwasser_P2_Ein := FALSE;
   E_Truebwasser_P2_St := FALSE;
   E_Truebwasser_P2_Bed_vOrt := FALSE;
   E_Truebwasser_P2_Bed_Fern := TRUE;
   E_Truebwasser_P2_AF_St := FALSE;
   E_Schlamm_AS_EA := FALSE;
   E_Schlamm_AS_EZ := TRUE;
   E_Schlamm_AS_St := FALSE;
   E_Schlamm_AS_Bed_vOrt := FALSE;
   E_Schlamm_AS_Bed_Fern := TRUE;
   E_Schlamm_AS_AF_St := FALSE;
   E_ZEN_Res_42_6 := FALSE;
   E_ZEN_Res_42_7 := FALSE;
   E_Schlamm_Besch_DF_ZI := FALSE;
   E_Schlamm_Besch_DF_St := FALSE;
   E_Truebwasser_Niv_St := FALSE;
   E_Truebwasser_DF_ZI := FALSE;
   E_Truebwasser_DF_St := FALSE;
   E_ZEN_Res_43_5 := FALSE;
   E_ZEN_Res_43_6 := FALSE;
   E_ZEN_Res_43_7 := FALSE;
   A_Schlamm_BP_Ein := FALSE;
   A_Truebwasser_P1_Ein := FALSE;
   A_Truebwasser_P2_Ein := FALSE;
   A_Schlamm_AS_Auf := FALSE;
   A_Schlamm_AS_Zu := FALSE;
   A_ZEN_Res_40_5 := FALSE;
   A_ZEN_Res_40_6 := FALSE;
   A_ZEN_Res_40_7 := FALSE;
   A_ZEN_Res_41_0 := FALSE;
   A_ZEN_Res_41_1 := FALSE;
   A_ZEN_Res_41_2 := FALSE;
   A_ZEN_Res_41_3 := FALSE;
   A_ZEN_Res_41_4 := FALSE;
   A_ZEN_Res_41_5 := FALSE;
   A_ZEN_Res_41_6 := FALSE;
   A_ZEN_Res_41_7 := FALSE;
   A_ZEN_Res_42_0 := FALSE;
   A_ZEN_Res_42_1 := FALSE;
   A_ZEN_Res_42_2 := FALSE;
   A_ZEN_Res_42_3 := FALSE;
   A_ZEN_Res_42_4 := FALSE;
   A_ZEN_Res_42_5 := FALSE;
   A_ZEN_Res_42_6 := FALSE;
   A_ZEN_Res_42_7 := FALSE;
   A_ZEN_Res_43_0 := FALSE;
   A_ZEN_Res_43_1 := FALSE;
   A_ZEN_Res_43_2 := FALSE;
   A_ZEN_Res_43_3 := FALSE;
   A_ZEN_Res_43_4 := FALSE;
   A_ZEN_Res_43_5 := FALSE;
   A_ZEN_Res_43_6 := FALSE;
   A_ZEN_Res_43_7 := FALSE;
   ZEN_DiagKom_IEC := FALSE;
   ZEN_DiagKom_DP_BF3 := FALSE;
   ZEN_DiagKom_DP_BF4 := FALSE;
   ZEN_DiagKom_DP_BF5 := FALSE;
   ZEN_DiagKom_DP_BF6 := FALSE;
   ZEN_DiagKom_DP_BF7 := FALSE;
   ZEN_DiagKom_DP_BF8 := FALSE;
   ZEN_DiagKom_DP_BF9 := FALSE;
   ZEN_DiagKom_DP_BF10 := FALSE;
   ZEN_DiagKom_DP_BF11 := FALSE;
   ZEN_DiagKom_DP_BF12 := FALSE;
   ZEN_DiagKom_DP_BF13 := FALSE;
   ZEN_DiagKom_DP_BF14 := FALSE;
   ZEN_DiagKom_DP_BF15 := FALSE;
   ZEN_DiagKom_DP_BF16 := FALSE;
   ZEN_DiagKom_DP_BF17 := FALSE;
   ZEN_ObjS_Begehung := FALSE;
   ZEN_ObjS_Alarm := FALSE;
   ZEN_ObjS_unscharf := FALSE;
   ZEN_ObjS_scharf := FALSE;
   ZEN_NA_res := FALSE;
   ZEN_Bed_aktiv := FALSE;
   ZEN_Res_DB100_40_6 := FALSE;
   ZEN_Res_DB100_40_7 := FALSE;
   BB_Auto_GeblW_G1_B1 := TRUE;
   BB_Auto_GeblW_G2_B2 := TRUE;
   BB_Auto_GeblW_G3_B1 := FALSE;
   BB_Auto_GeblW_G3_B2 := FALSE;
   ZEN_Res_DB100_41_4 := FALSE;
   ZEN_Res_DB100_41_5 := FALSE;
   ZEN_Res_DB100_41_6 := FALSE;
   ZEN_Res_DB100_41_7 := FALSE;
   Biocos1_BA_SU_RB := FALSE;
   Biocos1_BA_P1_RB := TRUE;
   Biocos1_BA_P2_RB := FALSE;
   Biocos1_BA_Aus_RB := FALSE;
   Biocos1_Auto_P1_aktiv := TRUE;
   Biocos1_Auto_P2_aktiv := FALSE;
   Biocos1_Auto_Bel_O2_Ein_RB := TRUE;
   Biocos1_Auto_Bel_O2_Aus_RB := FALSE;
   Biocos1_Auto_Bel_O2_St := FALSE;
   Biocos1_Auto_Bel_O2_min := FALSE;
   Biocos1_Auto_UeSS_Menge_Ein_RB := TRUE;
   Biocos1_Auto_UeSS_Menge_Aus_RB := FALSE;
   Biocos1_Auto_UeSS_Menge_St := FALSE;
   ZEN_Res_DB100_43_5 := FALSE;
   ZEN_Res_DB100_43_6 := FALSE;
   ZEN_Res_DB100_43_7 := FALSE;
   Biocos1_Auto_Bel_Phase := TRUE;
   Biocos1_Auto_Bel_Verz := FALSE;
   Biocos1_Auto_Bel_Frg := TRUE;
   Biocos1_Auto_Bel_Int := TRUE;
   Biocos1_Auto_UeSS := TRUE;
   ZEN_Res_DB100_44_5 := FALSE;
   ZEN_Res_DB100_44_6 := FALSE;
   ZEN_Res_DB100_44_7 := FALSE;
   Biocos1_Auto_U1 := FALSE;
   Biocos1_Auto_V1 := FALSE;
   Biocos1_Auto_A1 := TRUE;
   Biocos1_Auto_U2 := FALSE;
   Biocos1_Auto_V2 := TRUE;
   Biocos1_Auto_A2 := FALSE;
   Biocos1_Auto_SR1 := FALSE;
   Biocos1_Auto_SR2 := FALSE;
   Biocos2_BA_SU_RB := FALSE;
   Biocos2_BA_P1_RB := TRUE;
   Biocos2_BA_P2_RB := FALSE;
   Biocos2_BA_Aus_RB := FALSE;
   Biocos2_Auto_P1_aktiv := TRUE;
   Biocos2_Auto_P2_aktiv := FALSE;
   Biocos2_Auto_Bel_O2_Ein_RB := TRUE;
   Biocos2_Auto_Bel_O2_Aus_RB := FALSE;
   Biocos2_Auto_Bel_O2_St := FALSE;
   Biocos2_Auto_Bel_O2_min := FALSE;
   Biocos2_Auto_UeSS_Menge_Ein_RB := TRUE;
   Biocos2_Auto_UeSS_Menge_Aus_RB := FALSE;
   Biocos2_Auto_UeSS_Menge_St := FALSE;
   ZEN_Res_DB100_47_5 := FALSE;
   ZEN_Res_DB100_47_6 := FALSE;
   ZEN_Res_DB100_47_7 := FALSE;
   Biocos2_Auto_Bel_Phase := TRUE;
   Biocos2_Auto_Bel_Verz := FALSE;
   Biocos2_Auto_Bel_Frg := TRUE;
   Biocos2_Auto_Bel_Int := TRUE;
   Biocos2_Auto_UeSS := FALSE;
   ZEN_Res_DB100_48_5 := FALSE;
   ZEN_Res_DB100_48_6 := FALSE;
   ZEN_Res_DB100_48_7 := FALSE;
   Biocos2_Auto_U1 := FALSE;
   Biocos2_Auto_V1 := TRUE;
   Biocos2_Auto_A1 := FALSE;
   Biocos2_Auto_U2 := FALSE;
   Biocos2_Auto_V2 := FALSE;
   Biocos2_Auto_A2 := TRUE;
   Biocos2_Auto_SR1 := FALSE;
   Biocos2_Auto_SR2 := FALSE;
   ZEN_Res_DB100_50_0 := FALSE;
   ZEN_Res_DB100_50_1 := FALSE;
   ZEN_Res_DB100_50_2 := FALSE;
   ZEN_Res_DB100_50_3 := FALSE;
   ZEN_Res_DB100_50_4 := FALSE;
   ZEN_Res_DB100_50_5 := FALSE;
   ZEN_Res_DB100_50_6 := FALSE;
   ZEN_Res_DB100_50_7 := FALSE;
   ZEN_Res_DB100_51_0 := FALSE;
   ZEN_Res_DB100_51_1 := FALSE;
   ZEN_Res_DB100_51_2 := FALSE;
   ZEN_Res_DB100_51_3 := FALSE;
   ZEN_Res_DB100_51_4 := FALSE;
   ZEN_Res_DB100_51_5 := FALSE;
   ZEN_Res_DB100_51_6 := FALSE;
   ZEN_Res_DB100_51_7 := FALSE;
   IEC_Meld_LS_001 := FALSE;
   IEC_Meld_LS_002 := FALSE;
   IEC_Meld_LS_003 := FALSE;
   IEC_Meld_LS_004 := FALSE;
   IEC_Meld_LS_005 := FALSE;
   IEC_Meld_LS_006 := FALSE;
   IEC_Meld_LS_007 := FALSE;
   IEC_Meld_LS_008 := FALSE;
   IEC_Meld_LS_009 := FALSE;
   IEC_Meld_LS_010 := FALSE;
   IEC_Meld_LS_011 := FALSE;
   IEC_Meld_LS_012 := FALSE;
   IEC_Meld_LS_013 := FALSE;
   IEC_Meld_LS_014 := FALSE;
   IEC_Meld_LS_015 := FALSE;
   IEC_Meld_LS_016 := FALSE;
   IEC_Meld_LS_017 := FALSE;
   IEC_Meld_LS_018 := FALSE;
   IEC_Meld_LS_019 := FALSE;
   IEC_Meld_LS_020 := TRUE;
   IEC_Meld_LS_021 := FALSE;
   IEC_Meld_LS_022 := FALSE;
   IEC_Meld_LS_023 := FALSE;
   IEC_Meld_LS_024 := FALSE;
   IEC_Meld_LS_025 := FALSE;
   IEC_Meld_LS_026 := TRUE;
   IEC_Meld_LS_027 := FALSE;
   IEC_Meld_LS_028 := FALSE;
   IEC_Meld_LS_029 := FALSE;
   IEC_Meld_LS_030 := FALSE;
   IEC_Meld_LS_031 := FALSE;
   IEC_Meld_LS_032 := FALSE;
   Zulauf_PW_BA_Auto_RB := TRUE;
   Zulauf_PW_BA_Aus_RB := FALSE;
   Zulauf_PW_Auto_DF_max := FALSE;
   Zulauf_PW_Auto_Niv_max := FALSE;
   Zulauf_PW_Auto_Niv_AS := FALSE;
   Zulauf_PW_Auto_Niv_ZS := FALSE;
   Zulauf_PW_Auto_Niv_min := TRUE;
   Zulauf_PW_Auto_Frg_Ein := TRUE;
   Zulauf_PW_Auto_Frg_TeilAus := FALSE;
   Zulauf_PW_Auto_Frg_Aus := FALSE;
   ZEN_Res_DB100_57_2 := FALSE;
   Zulauf_RA_SA_Stillst := FALSE;
   ZEN_Res_DB100_57_4 := FALSE;
   ZEN_Res_DB100_57_5 := FALSE;
   ZEN_Res_DB100_57_6 := FALSE;
   ZEN_Res_DB100_57_7 := FALSE;
   Schlamm_TW_BA_Auto_RB := TRUE;
   Schlamm_TW_BA_Aus_RB := FALSE;
   Schlamm_TW_Auto_Frg_Zt := TRUE;
   Schlamm_TW_Auto_2P_Ein := FALSE;
   Schlamm_TW_Auto_1P_Ein := FALSE;
   ZEN_Res_DB100_58_5 := FALSE;
   ZEN_Res_DB100_58_6 := FALSE;
   ZEN_Res_DB100_58_7 := FALSE;
   Schlamm_Besch_BA_Auto_RB := FALSE;
   Schlamm_Besch_BA_Aus_RB := TRUE;
   Schlamm_Besch_Auto_Zt_max := FALSE;
   ZEN_Res_DB100_59_3 := FALSE;
   ZEN_Res_DB100_59_4 := FALSE;
   ZEN_Res_DB100_59_5 := FALSE;
   ZEN_Res_DB100_59_6 := FALSE;
   ZEN_Res_DB100_59_7 := FALSE;
   PO4_Elim_BA_Auto_RB := TRUE;
   PO4_Elim_BA_Hand_RB := FALSE;
   PO4_Elim_BA_Aus_RB := FALSE;
   PO4_Elim_Auto_P_Ein := TRUE;
   PO4_Elim_SC_Status_W1 := FALSE;
   PO4_Elim_SC_Status_W2 := FALSE;
   PO4_Elim_SC_Status_DevE := FALSE;
   PO4_Elim_SC_Status_CE := FALSE;
   Biocos1_BA_O2_Reg_FW_RB := FALSE;
   Biocos1_BA_O2_Reg_Auto_RB := TRUE;
   Biocos1_Auto_Bel_O2_Reg_St := FALSE;
   Biocos1_Auto_Bel_O2_Reg_GW_max := FALSE;
   ZEN_Res_DB100_61_4 := FALSE;
   ZEN_Res_DB100_61_5 := FALSE;
   ZEN_Res_DB100_61_6 := FALSE;
   ZEN_Res_DB100_61_7 := FALSE;
   Biocos2_BA_O2_Reg_FW_RB := FALSE;
   Biocos2_BA_O2_Reg_Auto_RB := TRUE;
   Biocos2_Auto_Bel_O2_Reg_St := FALSE;
   Biocos2_Auto_Bel_O2_Reg_GW_max := FALSE;
   ZEN_Res_DB100_62_4 := FALSE;
   ZEN_Res_DB100_62_5 := FALSE;
   ZEN_Res_DB100_62_6 := FALSE;
   ZEN_Res_DB100_62_7 := FALSE;
   ZEN_Res_DB100_63_0 := FALSE;
   ZEN_Res_DB100_63_1 := FALSE;
   ZEN_Res_DB100_63_2 := FALSE;
   ZEN_Res_DB100_63_3 := FALSE;
   ZEN_Res_DB100_63_4 := FALSE;
   ZEN_Res_DB100_63_5 := FALSE;
   ZEN_Res_DB100_63_6 := FALSE;
   ZEN_Res_DB100_63_7 := FALSE;
   BB_G1_KS_AM9 := FALSE;
   BB_G1_KS_AM10 := FALSE;
   BB_G1_KS_AM11 := FALSE;
   BB_G1_KS_AM12 := FALSE;
   BB_G1_KS_AM13 := FALSE;
   BB_G1_KS_AM14 := FALSE;
   BB_G1_KS_AM15 := FALSE;
   BB_G1_KS_AM16 := FALSE;
   BB_G1_KS_AM1 := FALSE;
   BB_G1_KS_AM2 := FALSE;
   BB_G1_KS_AM3 := FALSE;
   BB_G1_KS_AM4 := FALSE;
   BB_G1_KS_AM5 := FALSE;
   BB_G1_KS_AM6 := FALSE;
   BB_G1_KS_AM7 := FALSE;
   BB_G1_KS_AM8 := FALSE;
   BB_G1_KS_AM25 := FALSE;
   BB_G1_KS_AM26 := FALSE;
   BB_G1_KS_AM27 := FALSE;
   BB_G1_KS_AM28 := FALSE;
   BB_G1_KS_AM29 := FALSE;
   BB_G1_KS_AM30 := FALSE;
   BB_G1_KS_AM31 := FALSE;
   BB_G1_KS_AM32 := FALSE;
   BB_G1_KS_AM17 := FALSE;
   BB_G1_KS_AM18 := FALSE;
   BB_G1_KS_AM19 := FALSE;
   BB_G1_KS_AM20 := FALSE;
   BB_G1_KS_AM21 := FALSE;
   BB_G1_KS_AM22 := FALSE;
   BB_G1_KS_AM23 := FALSE;
   BB_G1_KS_AM24 := FALSE;
   BB_G1_KS_AM41 := FALSE;
   BB_G1_KS_AM42 := FALSE;
   BB_G1_KS_AM43 := FALSE;
   BB_G1_KS_AM44 := FALSE;
   BB_G1_KS_AM45 := FALSE;
   BB_G1_KS_AM46 := FALSE;
   BB_G1_KS_AM47 := FALSE;
   BB_G1_KS_AM48 := FALSE;
   BB_G1_KS_AM33 := FALSE;
   BB_G1_KS_AM34 := FALSE;
   BB_G1_KS_AM35 := FALSE;
   BB_G1_KS_AM36 := FALSE;
   BB_G1_KS_AM37 := FALSE;
   BB_G1_KS_AM38 := FALSE;
   BB_G1_KS_AM39 := FALSE;
   BB_G1_KS_AM40 := FALSE;
   BB_G1_KS_AM57 := FALSE;
   BB_G1_KS_AM58 := FALSE;
   BB_G1_KS_AM59 := FALSE;
   BB_G1_KS_AM60 := FALSE;
   BB_G1_KS_AM61 := FALSE;
   BB_G1_KS_AM62 := FALSE;
   BB_G1_KS_AM63 := FALSE;
   BB_G1_KS_AM64 := FALSE;
   BB_G1_KS_AM49 := FALSE;
   BB_G1_KS_AM50 := FALSE;
   BB_G1_KS_AM51 := FALSE;
   BB_G1_KS_AM52 := FALSE;
   BB_G1_KS_AM53 := FALSE;
   BB_G1_KS_AM54 := FALSE;
   BB_G1_KS_AM55 := FALSE;
   BB_G1_KS_AM56 := FALSE;
   BB_G1_KS_AM73 := FALSE;
   BB_G1_KS_AM74 := FALSE;
   BB_G1_KS_AM75 := FALSE;
   BB_G1_KS_AM76 := FALSE;
   BB_G1_KS_AM77 := FALSE;
   BB_G1_KS_AM78 := FALSE;
   BB_G1_KS_AM79 := FALSE;
   BB_G1_KS_AM80 := FALSE;
   BB_G1_KS_AM65 := FALSE;
   BB_G1_KS_AM66 := FALSE;
   BB_G1_KS_AM67 := FALSE;
   BB_G1_KS_AM68 := FALSE;
   BB_G1_KS_AM69 := FALSE;
   BB_G1_KS_AM70 := FALSE;
   BB_G1_KS_AM71 := FALSE;
   BB_G1_KS_AM72 := FALSE;
   BB_G1_KS_WM9 := FALSE;
   BB_G1_KS_WM10 := FALSE;
   BB_G1_KS_WM11 := FALSE;
   BB_G1_KS_WM12 := FALSE;
   BB_G1_KS_WM13 := FALSE;
   BB_G1_KS_WM14 := FALSE;
   BB_G1_KS_WM15 := FALSE;
   BB_G1_KS_WM16 := FALSE;
   BB_G1_KS_WM1 := FALSE;
   BB_G1_KS_WM2 := FALSE;
   BB_G1_KS_WM3 := FALSE;
   BB_G1_KS_WM4 := FALSE;
   BB_G1_KS_WM5 := FALSE;
   BB_G1_KS_WM6 := FALSE;
   BB_G1_KS_WM7 := FALSE;
   BB_G1_KS_WM8 := FALSE;
   BB_G1_KS_WM25 := FALSE;
   BB_G1_KS_WM26 := FALSE;
   BB_G1_KS_WM27 := FALSE;
   BB_G1_KS_WM28 := FALSE;
   BB_G1_KS_WM29 := FALSE;
   BB_G1_KS_WM30 := FALSE;
   BB_G1_KS_WM31 := FALSE;
   BB_G1_KS_WM32 := FALSE;
   BB_G1_KS_WM17 := FALSE;
   BB_G1_KS_WM18 := FALSE;
   BB_G1_KS_WM19 := FALSE;
   BB_G1_KS_WM20 := FALSE;
   BB_G1_KS_WM21 := FALSE;
   BB_G1_KS_WM22 := FALSE;
   BB_G1_KS_WM23 := FALSE;
   BB_G1_KS_WM24 := FALSE;
   BB_G1_KS_WM41 := FALSE;
   BB_G1_KS_WM42 := FALSE;
   BB_G1_KS_WM43 := FALSE;
   BB_G1_KS_WM44 := FALSE;
   BB_G1_KS_WM45 := FALSE;
   BB_G1_KS_WM46 := FALSE;
   BB_G1_KS_WM47 := FALSE;
   BB_G1_KS_WM48 := FALSE;
   BB_G1_KS_WM33 := FALSE;
   BB_G1_KS_WM34 := FALSE;
   BB_G1_KS_WM35 := FALSE;
   BB_G1_KS_WM36 := FALSE;
   BB_G1_KS_WM37 := FALSE;
   BB_G1_KS_WM38 := FALSE;
   BB_G1_KS_WM39 := FALSE;
   BB_G1_KS_WM40 := FALSE;
   BB_G1_KS_WM57 := FALSE;
   BB_G1_KS_WM58 := FALSE;
   BB_G1_KS_WM59 := FALSE;
   BB_G1_KS_WM60 := FALSE;
   BB_G1_KS_WM61 := FALSE;
   BB_G1_KS_WM62 := FALSE;
   BB_G1_KS_WM63 := FALSE;
   BB_G1_KS_WM64 := FALSE;
   BB_G1_KS_WM49 := FALSE;
   BB_G1_KS_WM50 := FALSE;
   BB_G1_KS_WM51 := FALSE;
   BB_G1_KS_WM52 := FALSE;
   BB_G1_KS_WM53 := FALSE;
   BB_G1_KS_WM54 := FALSE;
   BB_G1_KS_WM55 := FALSE;
   BB_G1_KS_WM56 := FALSE;
   BB_G1_KS_WM73 := FALSE;
   BB_G1_KS_WM74 := FALSE;
   BB_G1_KS_WM75 := FALSE;
   BB_G1_KS_WM76 := FALSE;
   BB_G1_KS_WM77 := FALSE;
   BB_G1_KS_WM78 := FALSE;
   BB_G1_KS_WM79 := FALSE;
   BB_G1_KS_WM80 := FALSE;
   BB_G1_KS_WM65 := FALSE;
   BB_G1_KS_WM66 := FALSE;
   BB_G1_KS_WM67 := FALSE;
   BB_G1_KS_WM68 := FALSE;
   BB_G1_KS_WM69 := FALSE;
   BB_G1_KS_WM70 := FALSE;
   BB_G1_KS_WM71 := FALSE;
   BB_G1_KS_WM72 := FALSE;
   BB_G1_KS_OM9 := FALSE;
   BB_G1_KS_OM10 := FALSE;
   BB_G1_KS_OM11 := FALSE;
   BB_G1_KS_OM12 := FALSE;
   BB_G1_KS_OM13 := FALSE;
   BB_G1_KS_OM14 := FALSE;
   BB_G1_KS_OM15 := FALSE;
   BB_G1_KS_OM16 := FALSE;
   BB_G1_KS_OM1 := FALSE;
   BB_G1_KS_OM2 := FALSE;
   BB_G1_KS_OM3 := FALSE;
   BB_G1_KS_OM4 := FALSE;
   BB_G1_KS_OM5 := FALSE;
   BB_G1_KS_OM6 := FALSE;
   BB_G1_KS_OM7 := FALSE;
   BB_G1_KS_OM8 := FALSE;
   BB_G1_KS_OM25 := FALSE;
   BB_G1_KS_OM26 := FALSE;
   BB_G1_KS_OM27 := FALSE;
   BB_G1_KS_OM28 := FALSE;
   BB_G1_KS_OM29 := FALSE;
   BB_G1_KS_OM30 := FALSE;
   BB_G1_KS_OM31 := FALSE;
   BB_G1_KS_OM32 := FALSE;
   BB_G1_KS_OM17 := FALSE;
   BB_G1_KS_OM18 := FALSE;
   BB_G1_KS_OM19 := FALSE;
   BB_G1_KS_OM20 := FALSE;
   BB_G1_KS_OM21 := FALSE;
   BB_G1_KS_OM22 := FALSE;
   BB_G1_KS_OM23 := FALSE;
   BB_G1_KS_OM24 := FALSE;
   BB_G1_KS_OM41 := FALSE;
   BB_G1_KS_OM42 := FALSE;
   BB_G1_KS_OM43 := FALSE;
   BB_G1_KS_OM44 := FALSE;
   BB_G1_KS_OM45 := FALSE;
   BB_G1_KS_OM46 := FALSE;
   BB_G1_KS_OM47 := FALSE;
   BB_G1_KS_OM48 := FALSE;
   BB_G1_KS_OM33 := FALSE;
   BB_G1_KS_OM34 := FALSE;
   BB_G1_KS_OM35 := FALSE;
   BB_G1_KS_OM36 := FALSE;
   BB_G1_KS_OM37 := FALSE;
   BB_G1_KS_OM38 := FALSE;
   BB_G1_KS_OM39 := FALSE;
   BB_G1_KS_OM40 := FALSE;
   BB_G1_KS_BS8 := FALSE;
   BB_G1_KS_BS9 := TRUE;
   BB_G1_KS_BS10 := FALSE;
   BB_G1_KS_BS11 := TRUE;
   BB_G1_KS_BS12 := FALSE;
   BB_G1_KS_BS13 := FALSE;
   BB_G1_KS_BS14 := FALSE;
   BB_G1_KS_BS15 := FALSE;
   BB_G1_KS_BS0 := TRUE;
   BB_G1_KS_BS1 := TRUE;
   BB_G1_KS_BS2 := TRUE;
   BB_G1_KS_BS3 := FALSE;
   BB_G1_KS_BS4 := FALSE;
   BB_G1_KS_BS5 := TRUE;
   BB_G1_KS_BS6 := FALSE;
   BB_G1_KS_BS7 := FALSE;
   BB_G1_KS_BS24 := FALSE;
   BB_G1_KS_BS25 := FALSE;
   BB_G1_KS_BS26 := FALSE;
   BB_G1_KS_BS27 := FALSE;
   BB_G1_KS_BS28 := FALSE;
   BB_G1_KS_BS29 := FALSE;
   BB_G1_KS_BS30 := FALSE;
   BB_G1_KS_BS31 := FALSE;
   BB_G1_KS_BS16 := TRUE;
   BB_G1_KS_BS17 := FALSE;
   BB_G1_KS_BS18 := FALSE;
   BB_G1_KS_BS19 := FALSE;
   BB_G1_KS_BS20 := FALSE;
   BB_G1_KS_BS21 := TRUE;
   BB_G1_KS_BS22 := FALSE;
   BB_G1_KS_BS23 := FALSE;
   BB_G1_KS_BS40 := FALSE;
   BB_G1_KS_BS41 := FALSE;
   BB_G1_KS_BS42 := FALSE;
   BB_G1_KS_BS43 := FALSE;
   BB_G1_KS_BS44 := FALSE;
   BB_G1_KS_BS45 := FALSE;
   BB_G1_KS_BS46 := FALSE;
   BB_G1_KS_BS47 := FALSE;
   BB_G1_KS_BS32 := FALSE;
   BB_G1_KS_BS33 := FALSE;
   BB_G1_KS_BS34 := FALSE;
   BB_G1_KS_BS35 := FALSE;
   BB_G1_KS_BS36 := FALSE;
   BB_G1_KS_BS37 := FALSE;
   BB_G1_KS_BS38 := FALSE;
   BB_G1_KS_BS39 := FALSE;
   BB_G1_KS_BS56 := FALSE;
   BB_G1_KS_BS57 := FALSE;
   BB_G1_KS_BS58 := FALSE;
   BB_G1_KS_BS59 := FALSE;
   BB_G1_KS_BS60 := FALSE;
   BB_G1_KS_BS61 := FALSE;
   BB_G1_KS_BS62 := FALSE;
   BB_G1_KS_BS63 := FALSE;
   BB_G1_KS_BS48 := FALSE;
   BB_G1_KS_BS49 := FALSE;
   BB_G1_KS_BS50 := FALSE;
   BB_G1_KS_BS51 := TRUE;
   BB_G1_KS_BS52 := FALSE;
   BB_G1_KS_BS53 := FALSE;
   BB_G1_KS_BS54 := FALSE;
   BB_G1_KS_BS55 := FALSE;
   BB_G2_KS_AM9 := FALSE;
   BB_G2_KS_AM10 := FALSE;
   BB_G2_KS_AM11 := FALSE;
   BB_G2_KS_AM12 := FALSE;
   BB_G2_KS_AM13 := FALSE;
   BB_G2_KS_AM14 := FALSE;
   BB_G2_KS_AM15 := FALSE;
   BB_G2_KS_AM16 := FALSE;
   BB_G2_KS_AM1 := FALSE;
   BB_G2_KS_AM2 := FALSE;
   BB_G2_KS_AM3 := FALSE;
   BB_G2_KS_AM4 := FALSE;
   BB_G2_KS_AM5 := FALSE;
   BB_G2_KS_AM6 := FALSE;
   BB_G2_KS_AM7 := FALSE;
   BB_G2_KS_AM8 := FALSE;
   BB_G2_KS_AM25 := FALSE;
   BB_G2_KS_AM26 := FALSE;
   BB_G2_KS_AM27 := FALSE;
   BB_G2_KS_AM28 := FALSE;
   BB_G2_KS_AM29 := FALSE;
   BB_G2_KS_AM30 := FALSE;
   BB_G2_KS_AM31 := FALSE;
   BB_G2_KS_AM32 := FALSE;
   BB_G2_KS_AM17 := FALSE;
   BB_G2_KS_AM18 := FALSE;
   BB_G2_KS_AM19 := FALSE;
   BB_G2_KS_AM20 := FALSE;
   BB_G2_KS_AM21 := FALSE;
   BB_G2_KS_AM22 := FALSE;
   BB_G2_KS_AM23 := FALSE;
   BB_G2_KS_AM24 := FALSE;
   BB_G2_KS_AM41 := FALSE;
   BB_G2_KS_AM42 := FALSE;
   BB_G2_KS_AM43 := FALSE;
   BB_G2_KS_AM44 := FALSE;
   BB_G2_KS_AM45 := FALSE;
   BB_G2_KS_AM46 := FALSE;
   BB_G2_KS_AM47 := FALSE;
   BB_G2_KS_AM48 := FALSE;
   BB_G2_KS_AM33 := FALSE;
   BB_G2_KS_AM34 := FALSE;
   BB_G2_KS_AM35 := FALSE;
   BB_G2_KS_AM36 := FALSE;
   BB_G2_KS_AM37 := FALSE;
   BB_G2_KS_AM38 := FALSE;
   BB_G2_KS_AM39 := FALSE;
   BB_G2_KS_AM40 := FALSE;
   BB_G2_KS_AM57 := FALSE;
   BB_G2_KS_AM58 := FALSE;
   BB_G2_KS_AM59 := FALSE;
   BB_G2_KS_AM60 := FALSE;
   BB_G2_KS_AM61 := FALSE;
   BB_G2_KS_AM62 := FALSE;
   BB_G2_KS_AM63 := FALSE;
   BB_G2_KS_AM64 := FALSE;
   BB_G2_KS_AM49 := FALSE;
   BB_G2_KS_AM50 := FALSE;
   BB_G2_KS_AM51 := FALSE;
   BB_G2_KS_AM52 := FALSE;
   BB_G2_KS_AM53 := FALSE;
   BB_G2_KS_AM54 := FALSE;
   BB_G2_KS_AM55 := FALSE;
   BB_G2_KS_AM56 := FALSE;
   BB_G2_KS_AM73 := FALSE;
   BB_G2_KS_AM74 := FALSE;
   BB_G2_KS_AM75 := FALSE;
   BB_G2_KS_AM76 := FALSE;
   BB_G2_KS_AM77 := FALSE;
   BB_G2_KS_AM78 := FALSE;
   BB_G2_KS_AM79 := FALSE;
   BB_G2_KS_AM80 := FALSE;
   BB_G2_KS_AM65 := FALSE;
   BB_G2_KS_AM66 := FALSE;
   BB_G2_KS_AM67 := FALSE;
   BB_G2_KS_AM68 := FALSE;
   BB_G2_KS_AM69 := FALSE;
   BB_G2_KS_AM70 := FALSE;
   BB_G2_KS_AM71 := FALSE;
   BB_G2_KS_AM72 := FALSE;
   BB_G2_KS_WM9 := FALSE;
   BB_G2_KS_WM10 := FALSE;
   BB_G2_KS_WM11 := FALSE;
   BB_G2_KS_WM12 := FALSE;
   BB_G2_KS_WM13 := FALSE;
   BB_G2_KS_WM14 := FALSE;
   BB_G2_KS_WM15 := FALSE;
   BB_G2_KS_WM16 := FALSE;
   BB_G2_KS_WM1 := FALSE;
   BB_G2_KS_WM2 := FALSE;
   BB_G2_KS_WM3 := FALSE;
   BB_G2_KS_WM4 := FALSE;
   BB_G2_KS_WM5 := FALSE;
   BB_G2_KS_WM6 := FALSE;
   BB_G2_KS_WM7 := FALSE;
   BB_G2_KS_WM8 := FALSE;
   BB_G2_KS_WM25 := FALSE;
   BB_G2_KS_WM26 := FALSE;
   BB_G2_KS_WM27 := FALSE;
   BB_G2_KS_WM28 := FALSE;
   BB_G2_KS_WM29 := FALSE;
   BB_G2_KS_WM30 := FALSE;
   BB_G2_KS_WM31 := FALSE;
   BB_G2_KS_WM32 := FALSE;
   BB_G2_KS_WM17 := FALSE;
   BB_G2_KS_WM18 := FALSE;
   BB_G2_KS_WM19 := FALSE;
   BB_G2_KS_WM20 := FALSE;
   BB_G2_KS_WM21 := FALSE;
   BB_G2_KS_WM22 := FALSE;
   BB_G2_KS_WM23 := FALSE;
   BB_G2_KS_WM24 := FALSE;
   BB_G2_KS_WM41 := FALSE;
   BB_G2_KS_WM42 := FALSE;
   BB_G2_KS_WM43 := FALSE;
   BB_G2_KS_WM44 := FALSE;
   BB_G2_KS_WM45 := FALSE;
   BB_G2_KS_WM46 := FALSE;
   BB_G2_KS_WM47 := FALSE;
   BB_G2_KS_WM48 := FALSE;
   BB_G2_KS_WM33 := FALSE;
   BB_G2_KS_WM34 := FALSE;
   BB_G2_KS_WM35 := FALSE;
   BB_G2_KS_WM36 := FALSE;
   BB_G2_KS_WM37 := FALSE;
   BB_G2_KS_WM38 := FALSE;
   BB_G2_KS_WM39 := FALSE;
   BB_G2_KS_WM40 := FALSE;
   BB_G2_KS_WM57 := FALSE;
   BB_G2_KS_WM58 := FALSE;
   BB_G2_KS_WM59 := FALSE;
   BB_G2_KS_WM60 := FALSE;
   BB_G2_KS_WM61 := FALSE;
   BB_G2_KS_WM62 := FALSE;
   BB_G2_KS_WM63 := FALSE;
   BB_G2_KS_WM64 := FALSE;
   BB_G2_KS_WM49 := FALSE;
   BB_G2_KS_WM50 := FALSE;
   BB_G2_KS_WM51 := FALSE;
   BB_G2_KS_WM52 := FALSE;
   BB_G2_KS_WM53 := FALSE;
   BB_G2_KS_WM54 := FALSE;
   BB_G2_KS_WM55 := FALSE;
   BB_G2_KS_WM56 := FALSE;
   BB_G2_KS_WM73 := FALSE;
   BB_G2_KS_WM74 := FALSE;
   BB_G2_KS_WM75 := FALSE;
   BB_G2_KS_WM76 := FALSE;
   BB_G2_KS_WM77 := FALSE;
   BB_G2_KS_WM78 := FALSE;
   BB_G2_KS_WM79 := FALSE;
   BB_G2_KS_WM80 := FALSE;
   BB_G2_KS_WM65 := FALSE;
   BB_G2_KS_WM66 := FALSE;
   BB_G2_KS_WM67 := FALSE;
   BB_G2_KS_WM68 := FALSE;
   BB_G2_KS_WM69 := FALSE;
   BB_G2_KS_WM70 := FALSE;
   BB_G2_KS_WM71 := FALSE;
   BB_G2_KS_WM72 := FALSE;
   BB_G2_KS_OM9 := FALSE;
   BB_G2_KS_OM10 := FALSE;
   BB_G2_KS_OM11 := FALSE;
   BB_G2_KS_OM12 := FALSE;
   BB_G2_KS_OM13 := FALSE;
   BB_G2_KS_OM14 := FALSE;
   BB_G2_KS_OM15 := FALSE;
   BB_G2_KS_OM16 := FALSE;
   BB_G2_KS_OM1 := FALSE;
   BB_G2_KS_OM2 := FALSE;
   BB_G2_KS_OM3 := FALSE;
   BB_G2_KS_OM4 := FALSE;
   BB_G2_KS_OM5 := FALSE;
   BB_G2_KS_OM6 := FALSE;
   BB_G2_KS_OM7 := FALSE;
   BB_G2_KS_OM8 := FALSE;
   BB_G2_KS_OM25 := FALSE;
   BB_G2_KS_OM26 := FALSE;
   BB_G2_KS_OM27 := FALSE;
   BB_G2_KS_OM28 := FALSE;
   BB_G2_KS_OM29 := FALSE;
   BB_G2_KS_OM30 := FALSE;
   BB_G2_KS_OM31 := FALSE;
   BB_G2_KS_OM32 := FALSE;
   BB_G2_KS_OM17 := FALSE;
   BB_G2_KS_OM18 := FALSE;
   BB_G2_KS_OM19 := FALSE;
   BB_G2_KS_OM20 := FALSE;
   BB_G2_KS_OM21 := FALSE;
   BB_G2_KS_OM22 := FALSE;
   BB_G2_KS_OM23 := FALSE;
   BB_G2_KS_OM24 := FALSE;
   BB_G2_KS_OM41 := FALSE;
   BB_G2_KS_OM42 := FALSE;
   BB_G2_KS_OM43 := FALSE;
   BB_G2_KS_OM44 := FALSE;
   BB_G2_KS_OM45 := FALSE;
   BB_G2_KS_OM46 := FALSE;
   BB_G2_KS_OM47 := FALSE;
   BB_G2_KS_OM48 := FALSE;
   BB_G2_KS_OM33 := FALSE;
   BB_G2_KS_OM34 := FALSE;
   BB_G2_KS_OM35 := FALSE;
   BB_G2_KS_OM36 := FALSE;
   BB_G2_KS_OM37 := FALSE;
   BB_G2_KS_OM38 := FALSE;
   BB_G2_KS_OM39 := FALSE;
   BB_G2_KS_OM40 := FALSE;
   BB_G2_KS_BS8 := FALSE;
   BB_G2_KS_BS9 := TRUE;
   BB_G2_KS_BS10 := FALSE;
   BB_G2_KS_BS11 := TRUE;
   BB_G2_KS_BS12 := FALSE;
   BB_G2_KS_BS13 := FALSE;
   BB_G2_KS_BS14 := FALSE;
   BB_G2_KS_BS15 := FALSE;
   BB_G2_KS_BS0 := TRUE;
   BB_G2_KS_BS1 := TRUE;
   BB_G2_KS_BS2 := TRUE;
   BB_G2_KS_BS3 := FALSE;
   BB_G2_KS_BS4 := FALSE;
   BB_G2_KS_BS5 := TRUE;
   BB_G2_KS_BS6 := FALSE;
   BB_G2_KS_BS7 := FALSE;
   BB_G2_KS_BS24 := FALSE;
   BB_G2_KS_BS25 := FALSE;
   BB_G2_KS_BS26 := FALSE;
   BB_G2_KS_BS27 := FALSE;
   BB_G2_KS_BS28 := FALSE;
   BB_G2_KS_BS29 := FALSE;
   BB_G2_KS_BS30 := FALSE;
   BB_G2_KS_BS31 := FALSE;
   BB_G2_KS_BS16 := TRUE;
   BB_G2_KS_BS17 := FALSE;
   BB_G2_KS_BS18 := FALSE;
   BB_G2_KS_BS19 := FALSE;
   BB_G2_KS_BS20 := FALSE;
   BB_G2_KS_BS21 := TRUE;
   BB_G2_KS_BS22 := FALSE;
   BB_G2_KS_BS23 := FALSE;
   BB_G2_KS_BS40 := FALSE;
   BB_G2_KS_BS41 := FALSE;
   BB_G2_KS_BS42 := FALSE;
   BB_G2_KS_BS43 := FALSE;
   BB_G2_KS_BS44 := FALSE;
   BB_G2_KS_BS45 := FALSE;
   BB_G2_KS_BS46 := FALSE;
   BB_G2_KS_BS47 := FALSE;
   BB_G2_KS_BS32 := FALSE;
   BB_G2_KS_BS33 := FALSE;
   BB_G2_KS_BS34 := FALSE;
   BB_G2_KS_BS35 := FALSE;
   BB_G2_KS_BS36 := FALSE;
   BB_G2_KS_BS37 := FALSE;
   BB_G2_KS_BS38 := FALSE;
   BB_G2_KS_BS39 := FALSE;
   BB_G2_KS_BS56 := FALSE;
   BB_G2_KS_BS57 := FALSE;
   BB_G2_KS_BS58 := FALSE;
   BB_G2_KS_BS59 := FALSE;
   BB_G2_KS_BS60 := FALSE;
   BB_G2_KS_BS61 := FALSE;
   BB_G2_KS_BS62 := FALSE;
   BB_G2_KS_BS63 := FALSE;
   BB_G2_KS_BS48 := FALSE;
   BB_G2_KS_BS49 := FALSE;
   BB_G2_KS_BS50 := FALSE;
   BB_G2_KS_BS51 := TRUE;
   BB_G2_KS_BS52 := FALSE;
   BB_G2_KS_BS53 := FALSE;
   BB_G2_KS_BS54 := FALSE;
   BB_G2_KS_BS55 := FALSE;
   BB_G3_KS_AM9 := FALSE;
   BB_G3_KS_AM10 := FALSE;
   BB_G3_KS_AM11 := FALSE;
   BB_G3_KS_AM12 := FALSE;
   BB_G3_KS_AM13 := FALSE;
   BB_G3_KS_AM14 := FALSE;
   BB_G3_KS_AM15 := FALSE;
   BB_G3_KS_AM16 := FALSE;
   BB_G3_KS_AM1 := FALSE;
   BB_G3_KS_AM2 := FALSE;
   BB_G3_KS_AM3 := FALSE;
   BB_G3_KS_AM4 := FALSE;
   BB_G3_KS_AM5 := FALSE;
   BB_G3_KS_AM6 := FALSE;
   BB_G3_KS_AM7 := FALSE;
   BB_G3_KS_AM8 := FALSE;
   BB_G3_KS_AM25 := FALSE;
   BB_G3_KS_AM26 := FALSE;
   BB_G3_KS_AM27 := FALSE;
   BB_G3_KS_AM28 := FALSE;
   BB_G3_KS_AM29 := FALSE;
   BB_G3_KS_AM30 := FALSE;
   BB_G3_KS_AM31 := FALSE;
   BB_G3_KS_AM32 := FALSE;
   BB_G3_KS_AM17 := FALSE;
   BB_G3_KS_AM18 := FALSE;
   BB_G3_KS_AM19 := FALSE;
   BB_G3_KS_AM20 := FALSE;
   BB_G3_KS_AM21 := FALSE;
   BB_G3_KS_AM22 := FALSE;
   BB_G3_KS_AM23 := FALSE;
   BB_G3_KS_AM24 := FALSE;
   BB_G3_KS_AM41 := FALSE;
   BB_G3_KS_AM42 := FALSE;
   BB_G3_KS_AM43 := FALSE;
   BB_G3_KS_AM44 := FALSE;
   BB_G3_KS_AM45 := FALSE;
   BB_G3_KS_AM46 := FALSE;
   BB_G3_KS_AM47 := FALSE;
   BB_G3_KS_AM48 := FALSE;
   BB_G3_KS_AM33 := FALSE;
   BB_G3_KS_AM34 := FALSE;
   BB_G3_KS_AM35 := FALSE;
   BB_G3_KS_AM36 := FALSE;
   BB_G3_KS_AM37 := FALSE;
   BB_G3_KS_AM38 := FALSE;
   BB_G3_KS_AM39 := FALSE;
   BB_G3_KS_AM40 := FALSE;
   BB_G3_KS_AM57 := FALSE;
   BB_G3_KS_AM58 := FALSE;
   BB_G3_KS_AM59 := FALSE;
   BB_G3_KS_AM60 := FALSE;
   BB_G3_KS_AM61 := FALSE;
   BB_G3_KS_AM62 := FALSE;
   BB_G3_KS_AM63 := FALSE;
   BB_G3_KS_AM64 := FALSE;
   BB_G3_KS_AM49 := FALSE;
   BB_G3_KS_AM50 := FALSE;
   BB_G3_KS_AM51 := FALSE;
   BB_G3_KS_AM52 := FALSE;
   BB_G3_KS_AM53 := FALSE;
   BB_G3_KS_AM54 := FALSE;
   BB_G3_KS_AM55 := FALSE;
   BB_G3_KS_AM56 := FALSE;
   BB_G3_KS_AM73 := FALSE;
   BB_G3_KS_AM74 := FALSE;
   BB_G3_KS_AM75 := FALSE;
   BB_G3_KS_AM76 := FALSE;
   BB_G3_KS_AM77 := FALSE;
   BB_G3_KS_AM78 := FALSE;
   BB_G3_KS_AM79 := FALSE;
   BB_G3_KS_AM80 := FALSE;
   BB_G3_KS_AM65 := FALSE;
   BB_G3_KS_AM66 := FALSE;
   BB_G3_KS_AM67 := FALSE;
   BB_G3_KS_AM68 := FALSE;
   BB_G3_KS_AM69 := FALSE;
   BB_G3_KS_AM70 := FALSE;
   BB_G3_KS_AM71 := FALSE;
   BB_G3_KS_AM72 := FALSE;
   BB_G3_KS_WM9 := FALSE;
   BB_G3_KS_WM10 := FALSE;
   BB_G3_KS_WM11 := FALSE;
   BB_G3_KS_WM12 := FALSE;
   BB_G3_KS_WM13 := FALSE;
   BB_G3_KS_WM14 := FALSE;
   BB_G3_KS_WM15 := FALSE;
   BB_G3_KS_WM16 := FALSE;
   BB_G3_KS_WM1 := FALSE;
   BB_G3_KS_WM2 := FALSE;
   BB_G3_KS_WM3 := FALSE;
   BB_G3_KS_WM4 := FALSE;
   BB_G3_KS_WM5 := FALSE;
   BB_G3_KS_WM6 := FALSE;
   BB_G3_KS_WM7 := FALSE;
   BB_G3_KS_WM8 := FALSE;
   BB_G3_KS_WM25 := FALSE;
   BB_G3_KS_WM26 := FALSE;
   BB_G3_KS_WM27 := FALSE;
   BB_G3_KS_WM28 := FALSE;
   BB_G3_KS_WM29 := FALSE;
   BB_G3_KS_WM30 := FALSE;
   BB_G3_KS_WM31 := FALSE;
   BB_G3_KS_WM32 := FALSE;
   BB_G3_KS_WM17 := FALSE;
   BB_G3_KS_WM18 := FALSE;
   BB_G3_KS_WM19 := FALSE;
   BB_G3_KS_WM20 := FALSE;
   BB_G3_KS_WM21 := FALSE;
   BB_G3_KS_WM22 := FALSE;
   BB_G3_KS_WM23 := FALSE;
   BB_G3_KS_WM24 := FALSE;
   BB_G3_KS_WM41 := FALSE;
   BB_G3_KS_WM42 := FALSE;
   BB_G3_KS_WM43 := FALSE;
   BB_G3_KS_WM44 := FALSE;
   BB_G3_KS_WM45 := FALSE;
   BB_G3_KS_WM46 := FALSE;
   BB_G3_KS_WM47 := FALSE;
   BB_G3_KS_WM48 := FALSE;
   BB_G3_KS_WM33 := FALSE;
   BB_G3_KS_WM34 := FALSE;
   BB_G3_KS_WM35 := FALSE;
   BB_G3_KS_WM36 := FALSE;
   BB_G3_KS_WM37 := FALSE;
   BB_G3_KS_WM38 := FALSE;
   BB_G3_KS_WM39 := FALSE;
   BB_G3_KS_WM40 := FALSE;
   BB_G3_KS_WM57 := FALSE;
   BB_G3_KS_WM58 := FALSE;
   BB_G3_KS_WM59 := FALSE;
   BB_G3_KS_WM60 := FALSE;
   BB_G3_KS_WM61 := FALSE;
   BB_G3_KS_WM62 := FALSE;
   BB_G3_KS_WM63 := FALSE;
   BB_G3_KS_WM64 := FALSE;
   BB_G3_KS_WM49 := FALSE;
   BB_G3_KS_WM50 := FALSE;
   BB_G3_KS_WM51 := FALSE;
   BB_G3_KS_WM52 := FALSE;
   BB_G3_KS_WM53 := FALSE;
   BB_G3_KS_WM54 := FALSE;
   BB_G3_KS_WM55 := FALSE;
   BB_G3_KS_WM56 := FALSE;
   BB_G3_KS_WM73 := FALSE;
   BB_G3_KS_WM74 := FALSE;
   BB_G3_KS_WM75 := FALSE;
   BB_G3_KS_WM76 := FALSE;
   BB_G3_KS_WM77 := FALSE;
   BB_G3_KS_WM78 := FALSE;
   BB_G3_KS_WM79 := FALSE;
   BB_G3_KS_WM80 := FALSE;
   BB_G3_KS_WM65 := FALSE;
   BB_G3_KS_WM66 := FALSE;
   BB_G3_KS_WM67 := FALSE;
   BB_G3_KS_WM68 := FALSE;
   BB_G3_KS_WM69 := FALSE;
   BB_G3_KS_WM70 := FALSE;
   BB_G3_KS_WM71 := FALSE;
   BB_G3_KS_WM72 := FALSE;
   BB_G3_KS_OM9 := FALSE;
   BB_G3_KS_OM10 := FALSE;
   BB_G3_KS_OM11 := FALSE;
   BB_G3_KS_OM12 := FALSE;
   BB_G3_KS_OM13 := FALSE;
   BB_G3_KS_OM14 := FALSE;
   BB_G3_KS_OM15 := FALSE;
   BB_G3_KS_OM16 := FALSE;
   BB_G3_KS_OM1 := FALSE;
   BB_G3_KS_OM2 := FALSE;
   BB_G3_KS_OM3 := FALSE;
   BB_G3_KS_OM4 := FALSE;
   BB_G3_KS_OM5 := FALSE;
   BB_G3_KS_OM6 := FALSE;
   BB_G3_KS_OM7 := FALSE;
   BB_G3_KS_OM8 := FALSE;
   BB_G3_KS_OM25 := FALSE;
   BB_G3_KS_OM26 := FALSE;
   BB_G3_KS_OM27 := FALSE;
   BB_G3_KS_OM28 := FALSE;
   BB_G3_KS_OM29 := FALSE;
   BB_G3_KS_OM30 := FALSE;
   BB_G3_KS_OM31 := FALSE;
   BB_G3_KS_OM32 := FALSE;
   BB_G3_KS_OM17 := FALSE;
   BB_G3_KS_OM18 := FALSE;
   BB_G3_KS_OM19 := FALSE;
   BB_G3_KS_OM20 := FALSE;
   BB_G3_KS_OM21 := FALSE;
   BB_G3_KS_OM22 := FALSE;
   BB_G3_KS_OM23 := FALSE;
   BB_G3_KS_OM24 := FALSE;
   BB_G3_KS_OM41 := FALSE;
   BB_G3_KS_OM42 := FALSE;
   BB_G3_KS_OM43 := FALSE;
   BB_G3_KS_OM44 := FALSE;
   BB_G3_KS_OM45 := FALSE;
   BB_G3_KS_OM46 := FALSE;
   BB_G3_KS_OM47 := FALSE;
   BB_G3_KS_OM48 := FALSE;
   BB_G3_KS_OM33 := FALSE;
   BB_G3_KS_OM34 := FALSE;
   BB_G3_KS_OM35 := FALSE;
   BB_G3_KS_OM36 := FALSE;
   BB_G3_KS_OM37 := FALSE;
   BB_G3_KS_OM38 := FALSE;
   BB_G3_KS_OM39 := FALSE;
   BB_G3_KS_OM40 := FALSE;
   BB_G3_KS_BS8 := FALSE;
   BB_G3_KS_BS9 := TRUE;
   BB_G3_KS_BS10 := FALSE;
   BB_G3_KS_BS11 := FALSE;
   BB_G3_KS_BS12 := FALSE;
   BB_G3_KS_BS13 := FALSE;
   BB_G3_KS_BS14 := FALSE;
   BB_G3_KS_BS15 := FALSE;
   BB_G3_KS_BS0 := TRUE;
   BB_G3_KS_BS1 := FALSE;
   BB_G3_KS_BS2 := FALSE;
   BB_G3_KS_BS3 := FALSE;
   BB_G3_KS_BS4 := FALSE;
   BB_G3_KS_BS5 := TRUE;
   BB_G3_KS_BS6 := FALSE;
   BB_G3_KS_BS7 := FALSE;
   BB_G3_KS_BS24 := FALSE;
   BB_G3_KS_BS25 := FALSE;
   BB_G3_KS_BS26 := FALSE;
   BB_G3_KS_BS27 := FALSE;
   BB_G3_KS_BS28 := FALSE;
   BB_G3_KS_BS29 := FALSE;
   BB_G3_KS_BS30 := FALSE;
   BB_G3_KS_BS31 := FALSE;
   BB_G3_KS_BS16 := TRUE;
   BB_G3_KS_BS17 := FALSE;
   BB_G3_KS_BS18 := FALSE;
   BB_G3_KS_BS19 := FALSE;
   BB_G3_KS_BS20 := TRUE;
   BB_G3_KS_BS21 := FALSE;
   BB_G3_KS_BS22 := FALSE;
   BB_G3_KS_BS23 := FALSE;
   BB_G3_KS_BS40 := FALSE;
   BB_G3_KS_BS41 := FALSE;
   BB_G3_KS_BS42 := FALSE;
   BB_G3_KS_BS43 := FALSE;
   BB_G3_KS_BS44 := FALSE;
   BB_G3_KS_BS45 := FALSE;
   BB_G3_KS_BS46 := FALSE;
   BB_G3_KS_BS47 := FALSE;
   BB_G3_KS_BS32 := FALSE;
   BB_G3_KS_BS33 := FALSE;
   BB_G3_KS_BS34 := FALSE;
   BB_G3_KS_BS35 := FALSE;
   BB_G3_KS_BS36 := FALSE;
   BB_G3_KS_BS37 := FALSE;
   BB_G3_KS_BS38 := FALSE;
   BB_G3_KS_BS39 := FALSE;
   BB_G3_KS_BS56 := FALSE;
   BB_G3_KS_BS57 := FALSE;
   BB_G3_KS_BS58 := FALSE;
   BB_G3_KS_BS59 := FALSE;
   BB_G3_KS_BS60 := FALSE;
   BB_G3_KS_BS61 := FALSE;
   BB_G3_KS_BS62 := FALSE;
   BB_G3_KS_BS63 := FALSE;
   BB_G3_KS_BS48 := FALSE;
   BB_G3_KS_BS49 := FALSE;
   BB_G3_KS_BS50 := FALSE;
   BB_G3_KS_BS51 := TRUE;
   BB_G3_KS_BS52 := FALSE;
   BB_G3_KS_BS53 := FALSE;
   BB_G3_KS_BS54 := FALSE;
   BB_G3_KS_BS55 := FALSE;

END_DATA_BLOCK

